LIN {X 0,Y 473.473,Z 413.056,A -85,B 0,C 180,E1 -7449.691,E2 -7449.691} C_VEL
LIN {X 0,Y 472.779,Z 426.431,A -85,B 0,C 180,E1 -7450.347,E2 -7450.347} C_VEL
LIN {X 0,Y 472.019,Z 440.423,A -85,B 0,C 180,E1 -7451.218,E2 -7451.218} C_VEL
LIN {X 0,Y 471.172,Z 453.208,A -85,B 0,C 180,E1 -7452.195,E2 -7452.195} C_VEL
LIN {X 0,Y 470.275,Z 466.134,A -85,B 0,C 180,E1 -7453.399,E2 -7453.399} C_VEL
LIN {X 0,Y 469.524,Z 476.835,A -85,B 0,C 180,E1 -7454.593,E2 -7454.593} C_VEL
LIN {X 0,Y 468.86,Z 486.774,A -85,B 0,C 180,E1 -7455.902,E2 -7455.902} C_VEL
LIN {X 0,Y 468.161,Z 496.122,A -85,B 0,C 180,E1 -7457.363,E2 -7457.363} C_VEL
LIN {X 0,Y 467.712,Z 504.564,A -85,B 0,C 180,E1 -7458.955,E2 -7458.955} C_VEL
LIN {X 0,Y 467.282,Z 511.235,A -85,B 0,C 180,E1 -7460.477,E2 -7460.477} C_VEL
LIN {X 0,Y 467.004,Z 517.412,A -85,B 0,C 180,E1 -7462.216,E2 -7462.216} C_VEL
LIN {X 0,Y 466.887,Z 522.181,A -85,B 0,C 180,E1 -7463.952,E2 -7463.952} C_VEL
LIN {X 0,Y 466.68,Z 525.681,A -85,B 0,C 180,E1 -7465.682,E2 -7465.682} C_VEL
LIN {X 0,Y 466.678,Z 527.994,A -85,B 0,C 180,E1 -7467.411,E2 -7467.411} C_VEL
LIN {X 0,Y 466.616,Z 529.179,A -85,B 0,C 180,E1 -7469.137,E2 -7469.137} C_VEL
LIN {X 0,Y 466.617,Z 529.196,A -85,B 0,C 180,E1 -7470.863,E2 -7470.863} C_VEL
LIN {X 0,Y 466.678,Z 528.081,A -85,B 0,C 180,E1 -7472.589,E2 -7472.589} C_VEL
LIN {X 0,Y 466.678,Z 525.836,A -85,B 0,C 180,E1 -7474.318,E2 -7474.318} C_VEL
LIN {X 0,Y 466.867,Z 522.401,A -85,B 0,C 180,E1 -7476.049,E2 -7476.049} C_VEL
LIN {X 0,Y 467.003,Z 517.703,A -85,B 0,C 180,E1 -7477.784,E2 -7477.784} C_VEL
LIN {X 0,Y 467.26,Z 511.612,A -85,B 0,C 180,E1 -7479.523,E2 -7479.523} C_VEL
LIN {X 0,Y 467.793,Z 503.938,A -85,B 0,C 180,E1 -7481.262,E2 -7481.262} C_VEL
LIN {X 0,Y 468.244,Z 495.615,A -85,B 0,C 180,E1 -7482.815,E2 -7482.815} C_VEL
LIN {X 0,Y 468.908,Z 485.901,A -85,B 0,C 180,E1 -7484.318,E2 -7484.318} C_VEL
LIN {X 0,Y 469.626,Z 475.791,A -85,B 0,C 180,E1 -7485.627,E2 -7485.627} C_VEL
LIN {X 0,Y 470.422,Z 464.385,A -85,B 0,C 180,E1 -7486.871,E2 -7486.871} C_VEL
LIN {X 0,Y 471.307,Z 451.682,A -85,B 0,C 180,E1 -7488.024,E2 -7488.024} C_VEL
LIN {X 0,Y 472.142,Z 438.564,A -85,B 0,C 180,E1 -7489.002,E2 -7489.002} C_VEL
LIN {X 0,Y 472.815,Z 426.069,A -85,B 0,C 180,E1 -7489.764,E2 -7489.764} C_VEL
LIN {X 0,Y 473.535,Z 411.357,A -85,B 0,C 180,E1 -7490.473,E2 -7490.473} C_VEL
LIN {X 0,Y 474.056,Z 395.831,A -85,B 0,C 180,E1 -7491.026,E2 -7491.026} C_VEL
LIN {X 0,Y 474.436,Z 382.034,A -85,B 0,C 180,E1 -7491.359,E2 -7491.359} C_VEL
LIN {X 0,Y 475.776,Z 266.855,A -85,B 0,C 180,E1 -7493.153,E2 -7493.153} C_VEL
LIN {X 0,Y 475.977,Z 239.419,A -85,B 0,C 180,E1 -7493.585,E2 -7493.585} C_VEL
LIN {X 0,Y 471.515,Z 220.798,A -85,B 0,C 180,E1 -7494.128,E2 -7494.128} C_VEL
LIN {X 0,Y 471.131,Z 219.52,A -85,B 0,C 180,E1 -7494.183,E2 -7494.183} C_VEL
LIN {X 0,Y 467.685,Z 203.856,A -85,B 0,C 180,E1 -7497.16,E2 -7497.16} C_VEL
LIN {X 0,Y 467.568,Z 203.868,A -85,B 0,C 180,E1 -7500.733,E2 -7500.733} C_VEL
LIN {X 0,Y 467.585,Z 203.866,A -85,B 0,C 180,E1 -7503.787,E2 -7503.787} C_VEL
LIN {X 0,Y 467.547,Z 203.87,A -85,B 0,C 180,E1 -7507.186,E2 -7507.186} C_VEL
LIN {X 0,Y 467.575,Z 203.862,A -85,B 0,C 180,E1 -7510.264,E2 -7510.264} C_VEL
LIN {X 0,Y 467.583,Z 203.863,A -85,B 0,C 180,E1 -7512.566,E2 -7512.566} C_VEL
LIN {X 0,Y 467.566,Z 203.868,A -85,B 0,C 180,E1 -7515.052,E2 -7515.052} C_VEL
LIN {X 0,Y 467.584,Z 203.86,A -85,B 0,C 180,E1 -7517.439,E2 -7517.439} C_VEL
LIN {X 0,Y 467.607,Z 203.863,A -85,B 0,C 180,E1 -7520.858,E2 -7520.858} C_VEL
LIN {X 0,Y 467.557,Z 203.864,A -85,B 0,C 180,E1 -7524.26,E2 -7524.26} C_VEL
LIN {X 0,Y 467.576,Z 203.858,A -85,B 0,C 180,E1 -7527.32,E2 -7527.32} C_VEL
LIN {X 0,Y 467.571,Z 203.863,A -85,B 0,C 180,E1 -7530.665,E2 -7530.665} C_VEL
LIN {X 0,Y 467.609,Z 203.861,A -85,B 0,C 180,E1 -7533.199,E2 -7533.199} C_VEL
LIN {X 0,Y 467.585,Z 203.864,A -85,B 0,C 180,E1 -7536.468,E2 -7536.468} C_VEL
LIN {X 0,Y 467.615,Z 203.858,A -85,B 0,C 180,E1 -7539.777,E2 -7539.777} C_VEL
LIN {X 0,Y 467.601,Z 203.86,A -85,B 0,C 180,E1 -7542.506,E2 -7542.506} C_VEL
LIN {X 0,Y 467.598,Z 203.859,A -85,B 0,C 180,E1 -7545.196,E2 -7545.196} C_VEL
LIN {X 0,Y 467.648,Z 203.854,A -85,B 0,C 180,E1 -7547.854,E2 -7547.854} C_VEL
LIN {X 0,Y 467.673,Z 203.852,A -85,B 0,C 180,E1 -7551.357,E2 -7551.357} C_VEL
LIN {X 0,Y 467.735,Z 203.842,A -85,B 0,C 180,E1 -7553.962,E2 -7553.962} C_VEL
LIN {X 0,Y 467.851,Z 203.829,A -85,B 0,C 180,E1 -7557.417,E2 -7557.417} C_VEL
LIN {X 0,Y 467.872,Z 203.822,A -85,B 0,C 180,E1 -7560,E2 -7560} C_VEL
LIN {X 0,Y 467.851,Z 203.834,A -85,B 0,C 180,E1 -7562.583,E2 -7562.583} C_VEL
LIN {X 0,Y 467.735,Z 203.845,A -85,B 0,C 180,E1 -7566.037,E2 -7566.037} C_VEL
LIN {X 0,Y 467.673,Z 203.853,A -85,B 0,C 180,E1 -7568.643,E2 -7568.643} C_VEL
LIN {X 0,Y 467.647,Z 203.858,A -85,B 0,C 180,E1 -7572.146,E2 -7572.146} C_VEL
LIN {X 0,Y 467.646,Z 203.856,A -85,B 0,C 180,E1 -7575.695,E2 -7575.695} C_VEL
LIN {X 0,Y 467.609,Z 203.864,A -85,B 0,C 180,E1 -7578.765,E2 -7578.765} C_VEL
LIN {X 0,Y 467.572,Z 203.861,A -85,B 0,C 180,E1 -7581.269,E2 -7581.269} C_VEL
LIN {X 0,Y 467.565,Z 203.869,A -85,B 0,C 180,E1 -7583.944,E2 -7583.944} C_VEL
LIN {X 0,Y 467.608,Z 203.862,A -85,B 0,C 180,E1 -7586.801,E2 -7586.801} C_VEL
LIN {X 0,Y 467.58,Z 203.865,A -85,B 0,C 180,E1 -7589.736,E2 -7589.736} C_VEL
LIN {X 0,Y 467.576,Z 203.862,A -85,B 0,C 180,E1 -7592.759,E2 -7592.759} C_VEL
LIN {X 0,Y 467.55,Z 203.871,A -85,B 0,C 180,E1 -7595.89,E2 -7595.89} C_VEL
LIN {X 0,Y 467.575,Z 203.86,A -85,B 0,C 180,E1 -7599.145,E2 -7599.145} C_VEL
LIN {X 0,Y 467.58,Z 203.865,A -85,B 0,C 180,E1 -7602.568,E2 -7602.568} C_VEL
LIN {X 0,Y 467.565,Z 203.865,A -85,B 0,C 180,E1 -7605.054,E2 -7605.054} C_VEL
LIN {X 0,Y 467.584,Z 203.864,A -85,B 0,C 180,E1 -7607.441,E2 -7607.441} C_VEL
LIN {X 0,Y 467.595,Z 203.861,A -85,B 0,C 180,E1 -7610.858,E2 -7610.858} C_VEL
LIN {X 0,Y 467.559,Z 203.869,A -85,B 0,C 180,E1 -7614.261,E2 -7614.261} C_VEL
LIN {X 0,Y 467.579,Z 203.868,A -85,B 0,C 180,E1 -7617.321,E2 -7617.321} C_VEL
LIN {X 0,Y 467.595,Z 203.901,A -85,B 0,C 180,E1 -7619.613,E2 -7619.613} C_VEL
LIN {X 0,Y 471.126,Z 218.42,A -85,B 0,C 180,E1 -7622.104,E2 -7622.104} C_VEL
LIN {X 0,Y 472.237,Z 223.722,A -85,B 0,C 180,E1 -7622.979,E2 -7622.979} C_VEL
LIN {X 0,Y 471.169,Z 243.147,A -85,B 0,C 180,E1 -7625.855,E2 -7625.855} C_VEL
LIN {X 0,Y 475.907,Z 268.042,A -85,B 0,C 180,E1 -7626.52,E2 -7626.52} C_VEL
LIN {X 0,Y 474.175,Z 410.193,A -85,B 0,C 180,E1 -7628.737,E2 -7628.737} C_VEL
LIN {X 0,Y 473.629,Z 425.893,A -85,B 0,C 180,E1 -7629.16,E2 -7629.16} C_VEL
LIN {X 0,Y 473.043,Z 439.94,A -85,B 0,C 180,E1 -7629.702,E2 -7629.702} C_VEL
LIN {X 0,Y 472.253,Z 454.431,A -85,B 0,C 180,E1 -7630.438,E2 -7630.438} C_VEL
LIN {X 0,Y 471.47,Z 467.941,A -85,B 0,C 180,E1 -7631.308,E2 -7631.308} C_VEL
LIN {X 0,Y 470.494,Z 481.695,A -85,B 0,C 180,E1 -7632.394,E2 -7632.394} C_VEL
LIN {X 0,Y 469.7,Z 494.151,A -85,B 0,C 180,E1 -7633.596,E2 -7633.596} C_VEL
LIN {X 0,Y 468.813,Z 506.366,A -85,B 0,C 180,E1 -7635.014,E2 -7635.014} C_VEL
LIN {X 0,Y 468.101,Z 517.231,A -85,B 0,C 180,E1 -7636.543,E2 -7636.543} C_VEL
LIN {X 0,Y 467.611,Z 526.284,A -85,B 0,C 180,E1 -7638.074,E2 -7638.074} C_VEL
LIN {X 0,Y 467.228,Z 533.793,A -85,B 0,C 180,E1 -7639.601,E2 -7639.601} C_VEL
LIN {X 0,Y 466.908,Z 540.8,A -85,B 0,C 180,E1 -7641.343,E2 -7641.343} C_VEL
LIN {X 0,Y 466.818,Z 546.314,A -85,B 0,C 180,E1 -7643.083,E2 -7643.083} C_VEL
LIN {X 0,Y 466.684,Z 550.48,A -85,B 0,C 180,E1 -7644.816,E2 -7644.816} C_VEL
LIN {X 0,Y 466.634,Z 553.402,A -85,B 0,C 180,E1 -7646.546,E2 -7646.546} C_VEL
LIN {X 0,Y 466.604,Z 555.144,A -85,B 0,C 180,E1 -7648.274,E2 -7648.274} C_VEL
LIN {X 0,Y 466.595,Z 555.742,A -85,B 0,C 180,E1 -7650,E2 -7650} C_VEL
LIN {X 0,Y 466.604,Z 555.142,A -85,B 0,C 180,E1 -7651.726,E2 -7651.726} C_VEL
LIN {X 0,Y 466.634,Z 553.396,A -85,B 0,C 180,E1 -7653.454,E2 -7653.454} C_VEL
LIN {X 0,Y 466.688,Z 550.477,A -85,B 0,C 180,E1 -7655.184,E2 -7655.184} C_VEL
LIN {X 0,Y 466.821,Z 546.316,A -85,B 0,C 180,E1 -7656.917,E2 -7656.917} C_VEL
LIN {X 0,Y 466.908,Z 540.799,A -85,B 0,C 180,E1 -7658.657,E2 -7658.657} C_VEL
LIN {X 0,Y 467.228,Z 533.783,A -85,B 0,C 180,E1 -7660.399,E2 -7660.399} C_VEL
LIN {X 0,Y 467.592,Z 526.274,A -85,B 0,C 180,E1 -7661.927,E2 -7661.927} C_VEL
LIN {X 0,Y 468.076,Z 517.225,A -85,B 0,C 180,E1 -7663.457,E2 -7663.457} C_VEL
LIN {X 0,Y 468.816,Z 506.356,A -85,B 0,C 180,E1 -7664.986,E2 -7664.986} C_VEL
LIN {X 0,Y 469.668,Z 494.142,A -85,B 0,C 180,E1 -7666.406,E2 -7666.406} C_VEL
LIN {X 0,Y 470.535,Z 481.688,A -85,B 0,C 180,E1 -7667.605,E2 -7667.605} C_VEL
LIN {X 0,Y 471.412,Z 469.438,A -85,B 0,C 180,E1 -7668.582,E2 -7668.582} C_VEL
LIN {X 0,Y 472.163,Z 456.21,A -85,B 0,C 180,E1 -7669.453,E2 -7669.453} C_VEL
LIN {X 0,Y 472.927,Z 443.069,A -85,B 0,C 180,E1 -7670.146,E2 -7670.146} C_VEL
LIN {X 0,Y 473.573,Z 427.912,A -85,B 0,C 180,E1 -7670.766,E2 -7670.766} C_VEL
LIN {X 0,Y 474.066,Z 412.397,A -85,B 0,C 180,E1 -7671.212,E2 -7671.212} C_VEL
LIN {X 0,Y 474.424,Z 390.321,A -85,B 0,C 180,E1 -7671.594,E2 -7671.594} C_VEL
LIN {X 0,Y 475.907,Z 267.885,A -85,B 0,C 180,E1 -7673.48,E2 -7673.48} C_VEL
LIN {X 0,Y 471.138,Z 243.171,A -85,B 0,C 180,E1 -7674.139,E2 -7674.139} C_VEL
LIN {X 0,Y 472.159,Z 225.592,A -85,B 0,C 180,E1 -7676.736,E2 -7676.736} C_VEL
LIN {X 0,Y 471.99,Z 222.192,A -85,B 0,C 180,E1 -7677.264,E2 -7677.264} C_VEL
LIN {X 0,Y 468.627,Z 208.028,A -85,B 0,C 180,E1 -7679.662,E2 -7679.662} C_VEL
LIN {X 0,Y 467.557,Z 203.866,A -85,B 0,C 180,E1 -7680.421,E2 -7680.421} C_VEL
LIN {X 0,Y 467.58,Z 203.857,A -85,B 0,C 180,E1 -7682.758,E2 -7682.758} C_VEL
LIN {X 0,Y 467.552,Z 203.869,A -85,B 0,C 180,E1 -7685.889,E2 -7685.889} C_VEL
LIN {X 0,Y 467.595,Z 203.862,A -85,B 0,C 180,E1 -7689.142,E2 -7689.142} C_VEL
LIN {X 0,Y 467.581,Z 203.863,A -85,B 0,C 180,E1 -7692.566,E2 -7692.566} C_VEL
LIN {X 0,Y 467.565,Z 203.863,A -85,B 0,C 180,E1 -7695.052,E2 -7695.052} C_VEL
LIN {X 0,Y 467.583,Z 203.862,A -85,B 0,C 180,E1 -7697.439,E2 -7697.439} C_VEL
LIN {X 0,Y 467.593,Z 203.859,A -85,B 0,C 180,E1 -7700.856,E2 -7700.856} C_VEL
LIN {X 0,Y 467.556,Z 203.865,A -85,B 0,C 180,E1 -7704.26,E2 -7704.26} C_VEL
LIN {X 0,Y 467.575,Z 203.861,A -85,B 0,C 180,E1 -7707.32,E2 -7707.32} C_VEL
LIN {X 0,Y 467.57,Z 203.862,A -85,B 0,C 180,E1 -7710.665,E2 -7710.665} C_VEL
LIN {X 0,Y 467.608,Z 203.859,A -85,B 0,C 180,E1 -7713.199,E2 -7713.199} C_VEL
LIN {X 0,Y 467.584,Z 203.858,A -85,B 0,C 180,E1 -7716.468,E2 -7716.468} C_VEL
LIN {X 0,Y 467.615,Z 203.857,A -85,B 0,C 180,E1 -7719.777,E2 -7719.777} C_VEL
LIN {X 0,Y 467.6,Z 203.859,A -85,B 0,C 180,E1 -7722.507,E2 -7722.507} C_VEL
LIN {X 0,Y 467.597,Z 203.862,A -85,B 0,C 180,E1 -7725.196,E2 -7725.196} C_VEL
LIN {X 0,Y 467.647,Z 203.857,A -85,B 0,C 180,E1 -7727.854,E2 -7727.854} C_VEL
LIN {X 0,Y 467.673,Z 203.854,A -85,B 0,C 180,E1 -7731.357,E2 -7731.357} C_VEL
LIN {X 0,Y 467.735,Z 203.845,A -85,B 0,C 180,E1 -7733.963,E2 -7733.963} C_VEL
LIN {X 0,Y 467.851,Z 203.835,A -85,B 0,C 180,E1 -7737.417,E2 -7737.417} C_VEL
LIN {X 0,Y 467.873,Z 203.824,A -85,B 0,C 180,E1 -7740,E2 -7740} C_VEL
LIN {X 0,Y 467.851,Z 203.829,A -85,B 0,C 180,E1 -7742.583,E2 -7742.583} C_VEL
LIN {X 0,Y 467.738,Z 203.843,A -85,B 0,C 180,E1 -7746.038,E2 -7746.038} C_VEL
LIN {X 0,Y 467.674,Z 203.849,A -85,B 0,C 180,E1 -7748.643,E2 -7748.643} C_VEL
LIN {X 0,Y 467.648,Z 203.852,A -85,B 0,C 180,E1 -7752.146,E2 -7752.146} C_VEL
LIN {X 0,Y 467.63,Z 203.856,A -85,B 0,C 180,E1 -7755.695,E2 -7755.695} C_VEL
LIN {X 0,Y 467.609,Z 203.862,A -85,B 0,C 180,E1 -7758.765,E2 -7758.765} C_VEL
LIN {X 0,Y 467.572,Z 203.868,A -85,B 0,C 180,E1 -7761.269,E2 -7761.269} C_VEL
LIN {X 0,Y 467.565,Z 203.862,A -85,B 0,C 180,E1 -7763.944,E2 -7763.944} C_VEL
LIN {X 0,Y 467.608,Z 203.849,A -85,B 0,C 180,E1 -7766.801,E2 -7766.801} C_VEL
LIN {X 0,Y 467.581,Z 203.863,A -85,B 0,C 180,E1 -7769.736,E2 -7769.736} C_VEL
LIN {X 0,Y 467.577,Z 203.868,A -85,B 0,C 180,E1 -7772.759,E2 -7772.759} C_VEL
LIN {X 0,Y 467.551,Z 203.865,A -85,B 0,C 180,E1 -7775.89,E2 -7775.89} C_VEL
LIN {X 0,Y 467.577,Z 203.864,A -85,B 0,C 180,E1 -7779.145,E2 -7779.145} C_VEL
LIN {X 0,Y 467.582,Z 203.864,A -85,B 0,C 180,E1 -7782.568,E2 -7782.568} C_VEL
LIN {X 0,Y 467.567,Z 203.869,A -85,B 0,C 180,E1 -7785.054,E2 -7785.054} C_VEL
LIN {X 0,Y 467.585,Z 203.864,A -85,B 0,C 180,E1 -7787.441,E2 -7787.441} C_VEL
LIN {X 0,Y 467.579,Z 203.864,A -85,B 0,C 180,E1 -7790.856,E2 -7790.856} C_VEL
LIN {X 0,Y 467.557,Z 203.867,A -85,B 0,C 180,E1 -7794.262,E2 -7794.262} C_VEL
LIN {X 0,Y 467.58,Z 203.866,A -85,B 0,C 180,E1 -7797.322,E2 -7797.322} C_VEL
LIN {X 0,Y 467.569,Z 203.868,A -85,B 0,C 180,E1 -7800.668,E2 -7800.668} C_VEL
LIN {X 0,Y 467.686,Z 203.923,A -85,B 0,C 180,E1 -7802.952,E2 -7802.952} C_VEL
LIN {X 0,Y 470.94,Z 218.784,A -85,B 0,C 180,E1 -7805.771,E2 -7805.771} C_VEL
LIN {X 0,Y 471.099,Z 219.687,A -85,B 0,C 180,E1 -7805.924,E2 -7805.924} C_VEL
LIN {X 0,Y 473.398,Z 228.223,A -85,B 0,C 180,E1 -7806.189,E2 -7806.189} C_VEL
LIN {X 0,Y 476.069,Z 240.442,A -85,B 0,C 180,E1 -7806.53,E2 -7806.53} C_VEL
LIN {X 0,Y 475.647,Z 279.036,A -85,B 0,C 180,E1 -7807.129,E2 -7807.129} C_VEL
LIN {X 0,Y 475.039,Z 284.883,A -85,B 0,C 180,E1 -7807.192,E2 -7807.192} C_VEL
LIN {X 0,Y 469.524,Z 303.949,A -85,B 0,C 180,E1 -7807.216,E2 -7807.216} C_VEL
LIN {X 0,Y 468.797,Z 309.804,A -85,B 0,C 180,E1 -7807.274,E2 -7807.274} C_VEL
LIN {X 0,Y 467.794,Z 384.871,A -85,B 0,C 180,E1 -7808.467,E2 -7808.467} C_VEL
LIN {X 0,Y 467.377,Z 400.309,A -85,B 0,C 180,E1 -7808.888,E2 -7808.888} C_VEL
LIN {X 0,Y 466.813,Z 413.523,A -85,B 0,C 180,E1 -7809.399,E2 -7809.399} C_VEL
LIN {X 0,Y 466.116,Z 426.64,A -85,B 0,C 180,E1 -7810.054,E2 -7810.054} C_VEL
LIN {X 0,Y 465.29,Z 440.631,A -85,B 0,C 180,E1 -7810.936,E2 -7810.936} C_VEL
LIN {X 0,Y 464.382,Z 453.415,A -85,B 0,C 180,E1 -7811.926,E2 -7811.926} C_VEL
LIN {X 0,Y 463.524,Z 465.627,A -85,B 0,C 180,E1 -7813.074,E2 -7813.074} C_VEL
LIN {X 0,Y 462.659,Z 477.04,A -85,B 0,C 180,E1 -7814.358,E2 -7814.358} C_VEL
LIN {X 0,Y 461.948,Z 486.979,A -85,B 0,C 180,E1 -7815.687,E2 -7815.687} C_VEL
LIN {X 0,Y 461.146,Z 496.829,A -85,B 0,C 180,E1 -7817.26,E2 -7817.26} C_VEL
LIN {X 0,Y 460.731,Z 504.767,A -85,B 0,C 180,E1 -7818.785,E2 -7818.785} C_VEL
LIN {X 0,Y 460.259,Z 511.438,A -85,B 0,C 180,E1 -7820.331,E2 -7820.331} C_VEL
LIN {X 0,Y 459.963,Z 517.614,A -85,B 0,C 180,E1 -7822.096,E2 -7822.096} C_VEL
LIN {X 0,Y 459.816,Z 522.383,A -85,B 0,C 180,E1 -7823.858,E2 -7823.858} C_VEL
LIN {X 0,Y 459.594,Z 525.883,A -85,B 0,C 180,E1 -7825.615,E2 -7825.615} C_VEL
LIN {X 0,Y 459.6,Z 528.195,A -85,B 0,C 180,E1 -7827.371,E2 -7827.371} C_VEL
LIN {X 0,Y 459.52,Z 529.38,A -85,B 0,C 180,E1 -7829.124,E2 -7829.124} C_VEL
LIN {X 0,Y 459.521,Z 529.397,A -85,B 0,C 180,E1 -7830.876,E2 -7830.876} C_VEL
LIN {X 0,Y 459.6,Z 528.281,A -85,B 0,C 180,E1 -7832.629,E2 -7832.629} C_VEL
LIN {X 0,Y 459.592,Z 526.037,A -85,B 0,C 180,E1 -7834.385,E2 -7834.385} C_VEL
LIN {X 0,Y 459.794,Z 522.602,A -85,B 0,C 180,E1 -7836.142,E2 -7836.142} C_VEL
LIN {X 0,Y 459.962,Z 517.902,A -85,B 0,C 180,E1 -7837.904,E2 -7837.904} C_VEL
LIN {X 0,Y 460.231,Z 511.812,A -85,B 0,C 180,E1 -7839.67,E2 -7839.67} C_VEL
LIN {X 0,Y 460.8,Z 504.137,A -85,B 0,C 180,E1 -7841.436,E2 -7841.436} C_VEL
LIN {X 0,Y 461.26,Z 496.054,A -85,B 0,C 180,E1 -7842.97,E2 -7842.97} C_VEL
LIN {X 0,Y 461.994,Z 486.1,A -85,B 0,C 180,E1 -7844.537,E2 -7844.537} C_VEL
LIN {X 0,Y 462.737,Z 475.99,A -85,B 0,C 180,E1 -7845.865,E2 -7845.865} C_VEL
LIN {X 0,Y 463.578,Z 465.088,A -85,B 0,C 180,E1 -7847.073,E2 -7847.073} C_VEL
LIN {X 0,Y 464.459,Z 453.163,A -85,B 0,C 180,E1 -7848.185,E2 -7848.185} C_VEL
LIN {X 0,Y 465.312,Z 440.334,A -85,B 0,C 180,E1 -7849.178,E2 -7849.178} C_VEL
LIN {X 0,Y 466.155,Z 426.261,A -85,B 0,C 180,E1 -7850.059,E2 -7850.059} C_VEL
LIN {X 0,Y 466.902,Z 411.121,A -85,B 0,C 180,E1 -7850.796,E2 -7850.796} C_VEL
LIN {X 0,Y 467.477,Z 395.646,A -85,B 0,C 180,E1 -7851.349,E2 -7851.349} C_VEL
LIN {X 0,Y 467.857,Z 381.93,A -85,B 0,C 180,E1 -7851.68,E2 -7851.68} C_VEL
LIN {X 0,Y 469.426,Z 255.668,A -85,B 0,C 180,E1 -7853.67,E2 -7853.67} C_VEL
LIN {X 0,Y 469.433,Z 240.217,A -85,B 0,C 180,E1 -7853.923,E2 -7853.923} C_VEL
LIN {X 0,Y 465.221,Z 222.931,A -85,B 0,C 180,E1 -7854.443,E2 -7854.443} C_VEL
LIN {X 0,Y 463.984,Z 219.732,A -85,B 0,C 180,E1 -7854.58,E2 -7854.58} C_VEL
LIN {X 0,Y 460.94,Z 206.042,A -85,B 0,C 180,E1 -7857.22,E2 -7857.22} C_VEL
LIN {X 0,Y 460.592,Z 204.74,A -85,B 0,C 180,E1 -7857.491,E2 -7857.491} C_VEL
LIN {X 0,Y 460.509,Z 204.747,A -85,B 0,C 180,E1 -7860.239,E2 -7860.239} C_VEL
LIN {X 0,Y 460.527,Z 204.749,A -85,B 0,C 180,E1 -7863.324,E2 -7863.324} C_VEL
LIN {X 0,Y 460.475,Z 204.749,A -85,B 0,C 180,E1 -7866.528,E2 -7866.528} C_VEL
LIN {X 0,Y 460.542,Z 204.745,A -85,B 0,C 180,E1 -7868.897,E2 -7868.897} C_VEL
LIN {X 0,Y 460.52,Z 204.743,A -85,B 0,C 180,E1 -7872.18,E2 -7872.18} C_VEL
LIN {X 0,Y 460.512,Z 204.749,A -85,B 0,C 180,E1 -7875.411,E2 -7875.411} C_VEL
LIN {X 0,Y 460.53,Z 204.737,A -85,B 0,C 180,E1 -7878.396,E2 -7878.396} C_VEL
LIN {X 0,Y 460.536,Z 204.739,A -85,B 0,C 180,E1 -7881.268,E2 -7881.268} C_VEL
LIN {X 0,Y 460.508,Z 204.743,A -85,B 0,C 180,E1 -7884.554,E2 -7884.554} C_VEL
LIN {X 0,Y 460.526,Z 204.732,A -85,B 0,C 180,E1 -7887.715,E2 -7887.715} C_VEL
LIN {X 0,Y 460.54,Z 204.739,A -85,B 0,C 180,E1 -7890.769,E2 -7890.769} C_VEL
LIN {X 0,Y 460.555,Z 204.736,A -85,B 0,C 180,E1 -7893.734,E2 -7893.734} C_VEL
LIN {X 0,Y 460.538,Z 204.743,A -85,B 0,C 180,E1 -7896.623,E2 -7896.623} C_VEL
LIN {X 0,Y 460.544,Z 204.741,A -85,B 0,C 180,E1 -7899.452,E2 -7899.452} C_VEL
LIN {X 0,Y 460.551,Z 204.736,A -85,B 0,C 180,E1 -7902.23,E2 -7902.23} C_VEL
LIN {X 0,Y 460.557,Z 204.739,A -85,B 0,C 180,E1 -7904.964,E2 -7904.964} C_VEL
LIN {X 0,Y 460.604,Z 204.736,A -85,B 0,C 180,E1 -7908.559,E2 -7908.559} C_VEL
LIN {X 0,Y 460.686,Z 204.722,A -85,B 0,C 180,E1 -7912.108,E2 -7912.108} C_VEL
LIN {X 0,Y 460.689,Z 204.722,A -85,B 0,C 180,E1 -7914.748,E2 -7914.748} C_VEL
LIN {X 0,Y 460.816,Z 204.706,A -85,B 0,C 180,E1 -7917.377,E2 -7917.377} C_VEL
LIN {X 0,Y 460.843,Z 204.698,A -85,B 0,C 180,E1 -7920,E2 -7920} C_VEL
LIN {X 0,Y 460.816,Z 204.71,A -85,B 0,C 180,E1 -7922.622,E2 -7922.622} C_VEL
LIN {X 0,Y 460.701,Z 204.722,A -85,B 0,C 180,E1 -7926.13,E2 -7926.13} C_VEL
LIN {X 0,Y 460.62,Z 204.732,A -85,B 0,C 180,E1 -7928.776,E2 -7928.776} C_VEL
LIN {X 0,Y 460.604,Z 204.735,A -85,B 0,C 180,E1 -7932.445,E2 -7932.445} C_VEL
LIN {X 0,Y 460.613,Z 204.735,A -85,B 0,C 180,E1 -7936.007,E2 -7936.007} C_VEL
LIN {X 0,Y 460.561,Z 204.739,A -85,B 0,C 180,E1 -7939.616,E2 -7939.616} C_VEL
LIN {X 0,Y 460.503,Z 204.749,A -85,B 0,C 180,E1 -7942.429,E2 -7942.429} C_VEL
LIN {X 0,Y 460.559,Z 204.737,A -85,B 0,C 180,E1 -7945.802,E2 -7945.802} C_VEL
LIN {X 0,Y 460.55,Z 204.745,A -85,B 0,C 180,E1 -7948.233,E2 -7948.233} C_VEL
LIN {X 0,Y 460.517,Z 204.743,A -85,B 0,C 180,E1 -7951.284,E2 -7951.284} C_VEL
LIN {X 0,Y 460.527,Z 204.745,A -85,B 0,C 180,E1 -7954.507,E2 -7954.507} C_VEL
LIN {X 0,Y 460.495,Z 204.747,A -85,B 0,C 180,E1 -7957.624,E2 -7957.624} C_VEL
LIN {X 0,Y 460.535,Z 204.732,A -85,B 0,C 180,E1 -7960.27,E2 -7960.27} C_VEL
LIN {X 0,Y 460.494,Z 204.747,A -85,B 0,C 180,E1 -7963.376,E2 -7963.376} C_VEL
LIN {X 0,Y 460.495,Z 204.747,A -85,B 0,C 180,E1 -7966.625,E2 -7966.625} C_VEL
LIN {X 0,Y 460.553,Z 204.743,A -85,B 0,C 180,E1 -7969.729,E2 -7969.729} C_VEL
LIN {X 0,Y 460.524,Z 204.739,A -85,B 0,C 180,E1 -7972.52,E2 -7972.52} C_VEL
LIN {X 0,Y 460.545,Z 204.745,A -85,B 0,C 180,E1 -7975.625,E2 -7975.625} C_VEL
LIN {X 0,Y 460.534,Z 204.742,A -85,B 0,C 180,E1 -7978.745,E2 -7978.745} C_VEL
LIN {X 0,Y 460.566,Z 204.887,A -85,B 0,C 180,E1 -7979.289,E2 -7979.289} C_VEL
LIN {X 0,Y 464.003,Z 218.784,A -85,B 0,C 180,E1 -7981.726,E2 -7981.726} C_VEL
LIN {X 0,Y 465.427,Z 225.43,A -85,B 0,C 180,E1 -7982.846,E2 -7982.846} C_VEL
LIN {X 0,Y 464.373,Z 242.94,A -85,B 0,C 180,E1 -7985.478,E2 -7985.478} C_VEL
LIN {X 0,Y 469.382,Z 268.809,A -85,B 0,C 180,E1 -7986.189,E2 -7986.189} C_VEL
LIN {X 0,Y 467.581,Z 408.682,A -85,B 0,C 180,E1 -7988.393,E2 -7988.393} C_VEL
LIN {X 0,Y 467.101,Z 424.245,A -85,B 0,C 180,E1 -7988.804,E2 -7988.804} C_VEL
LIN {X 0,Y 466.417,Z 438.561,A -85,B 0,C 180,E1 -7989.348,E2 -7989.348} C_VEL
LIN {X 0,Y 465.651,Z 452.242,A -85,B 0,C 180,E1 -7990.034,E2 -7990.034} C_VEL
LIN {X 0,Y 464.751,Z 466.155,A -85,B 0,C 180,E1 -7990.913,E2 -7990.913} C_VEL
LIN {X 0,Y 463.845,Z 478.904,A -85,B 0,C 180,E1 -7991.905,E2 -7991.905} C_VEL
LIN {X 0,Y 462.924,Z 491.791,A -85,B 0,C 180,E1 -7993.12,E2 -7993.12} C_VEL
LIN {X 0,Y 462.119,Z 502.601,A -85,B 0,C 180,E1 -7994.339,E2 -7994.339} C_VEL
LIN {X 0,Y 461.427,Z 512.597,A -85,B 0,C 180,E1 -7995.67,E2 -7995.67} C_VEL
LIN {X 0,Y 460.768,Z 522.627,A -85,B 0,C 180,E1 -7997.268,E2 -7997.268} C_VEL
LIN {X 0,Y 460.392,Z 530.546,A -85,B 0,C 180,E1 -7998.777,E2 -7998.777} C_VEL
LIN {X 0,Y 459.939,Z 537.293,A -85,B 0,C 180,E1 -8000.324,E2 -8000.324} C_VEL
LIN {X 0,Y 459.765,Z 543.531,A -85,B 0,C 180,E1 -8002.093,E2 -8002.093} C_VEL
LIN {X 0,Y 459.617,Z 548.356,A -85,B 0,C 180,E1 -8003.856,E2 -8003.856} C_VEL
LIN {X 0,Y 459.517,Z 551.89,A -85,B 0,C 180,E1 -8005.614,E2 -8005.614} C_VEL
LIN {X 0,Y 459.573,Z 554.218,A -85,B 0,C 180,E1 -8007.371,E2 -8007.371} C_VEL
LIN {X 0,Y 459.519,Z 555.387,A -85,B 0,C 180,E1 -8009.124,E2 -8009.124} C_VEL
LIN {X 0,Y 459.519,Z 555.386,A -85,B 0,C 180,E1 -8010.876,E2 -8010.876} C_VEL
LIN {X 0,Y 459.573,Z 554.213,A -85,B 0,C 180,E1 -8012.629,E2 -8012.629} C_VEL
LIN {X 0,Y 459.517,Z 551.884,A -85,B 0,C 180,E1 -8014.386,E2 -8014.386} C_VEL
LIN {X 0,Y 459.64,Z 548.355,A -85,B 0,C 180,E1 -8016.144,E2 -8016.144} C_VEL
LIN {X 0,Y 459.765,Z 543.532,A -85,B 0,C 180,E1 -8017.907,E2 -8017.907} C_VEL
LIN {X 0,Y 459.939,Z 537.285,A -85,B 0,C 180,E1 -8019.676,E2 -8019.676} C_VEL
LIN {X 0,Y 460.392,Z 530.534,A -85,B 0,C 180,E1 -8021.223,E2 -8021.223} C_VEL
LIN {X 0,Y 460.733,Z 522.616,A -85,B 0,C 180,E1 -8022.733,E2 -8022.733} C_VEL
LIN {X 0,Y 461.429,Z 512.587,A -85,B 0,C 180,E1 -8024.329,E2 -8024.329} C_VEL
LIN {X 0,Y 462.137,Z 502.587,A -85,B 0,C 180,E1 -8025.66,E2 -8025.66} C_VEL
LIN {X 0,Y 462.948,Z 491.599,A -85,B 0,C 180,E1 -8026.898,E2 -8026.898} C_VEL
LIN {X 0,Y 463.866,Z 478.888,A -85,B 0,C 180,E1 -8028.095,E2 -8028.095} C_VEL
LIN {X 0,Y 464.807,Z 466.121,A -85,B 0,C 180,E1 -8029.085,E2 -8029.085} C_VEL
LIN {X 0,Y 465.667,Z 452.195,A -85,B 0,C 180,E1 -8029.966,E2 -8029.966} C_VEL
LIN {X 0,Y 466.424,Z 438.456,A -85,B 0,C 180,E1 -8030.654,E2 -8030.654} C_VEL
LIN {X 0,Y 467.087,Z 423.263,A -85,B 0,C 180,E1 -8031.226,E2 -8031.226} C_VEL
LIN {X 0,Y 467.579,Z 408.546,A -85,B 0,C 180,E1 -8031.607,E2 -8031.607} C_VEL
LIN {X 0,Y 469.38,Z 268.62,A -85,B 0,C 180,E1 -8033.811,E2 -8033.811} C_VEL
LIN {X 0,Y 464.401,Z 242.824,A -85,B 0,C 180,E1 -8034.533,E2 -8034.533} C_VEL
LIN {X 0,Y 465.383,Z 225.239,A -85,B 0,C 180,E1 -8037.181,E2 -8037.181} C_VEL
LIN {X 0,Y 462.596,Z 212.985,A -85,B 0,C 180,E1 -8039.272,E2 -8039.272} C_VEL
LIN {X 0,Y 460.544,Z 204.738,A -85,B 0,C 180,E1 -8040.744,E2 -8040.744} C_VEL
LIN {X 0,Y 460.526,Z 204.734,A -85,B 0,C 180,E1 -8043.324,E2 -8043.324} C_VEL
LIN {X 0,Y 460.475,Z 204.751,A -85,B 0,C 180,E1 -8046.529,E2 -8046.529} C_VEL
LIN {X 0,Y 460.57,Z 204.741,A -85,B 0,C 180,E1 -8049.857,E2 -8049.857} C_VEL
LIN {X 0,Y 460.508,Z 204.743,A -85,B 0,C 180,E1 -8052.9,E2 -8052.9} C_VEL
LIN {X 0,Y 460.506,Z 204.748,A -85,B 0,C 180,E1 -8055.83,E2 -8055.83} C_VEL
LIN {X 0,Y 460.533,Z 204.738,A -85,B 0,C 180,E1 -8058.989,E2 -8058.989} C_VEL
LIN {X 0,Y 460.533,Z 204.74,A -85,B 0,C 180,E1 -8061.268,E2 -8061.268} C_VEL
LIN {X 0,Y 460.507,Z 204.741,A -85,B 0,C 180,E1 -8064.554,E2 -8064.554} C_VEL
LIN {X 0,Y 460.525,Z 204.743,A -85,B 0,C 180,E1 -8067.715,E2 -8067.715} C_VEL
LIN {X 0,Y 460.539,Z 204.737,A -85,B 0,C 180,E1 -8070.769,E2 -8070.769} C_VEL
LIN {X 0,Y 460.555,Z 204.741,A -85,B 0,C 180,E1 -8073.734,E2 -8073.734} C_VEL
LIN {X 0,Y 460.538,Z 204.736,A -85,B 0,C 180,E1 -8076.624,E2 -8076.624} C_VEL
LIN {X 0,Y 460.543,Z 204.732,A -85,B 0,C 180,E1 -8079.452,E2 -8079.452} C_VEL
LIN {X 0,Y 460.55,Z 204.739,A -85,B 0,C 180,E1 -8082.23,E2 -8082.23} C_VEL
LIN {X 0,Y 460.556,Z 204.738,A -85,B 0,C 180,E1 -8084.965,E2 -8084.965} C_VEL
LIN {X 0,Y 460.604,Z 204.73,A -85,B 0,C 180,E1 -8088.559,E2 -8088.559} C_VEL
LIN {X 0,Y 460.686,Z 204.721,A -85,B 0,C 180,E1 -8092.108,E2 -8092.108} C_VEL
LIN {X 0,Y 460.689,Z 204.721,A -85,B 0,C 180,E1 -8094.748,E2 -8094.748} C_VEL
LIN {X 0,Y 460.816,Z 204.71,A -85,B 0,C 180,E1 -8097.378,E2 -8097.378} C_VEL
LIN {X 0,Y 460.844,Z 204.699,A -85,B 0,C 180,E1 -8100,E2 -8100} C_VEL
LIN {X 0,Y 460.816,Z 204.706,A -85,B 0,C 180,E1 -8102.623,E2 -8102.623} C_VEL
LIN {X 0,Y 460.704,Z 204.719,A -85,B 0,C 180,E1 -8106.13,E2 -8106.13} C_VEL
LIN {X 0,Y 460.621,Z 204.728,A -85,B 0,C 180,E1 -8108.776,E2 -8108.776} C_VEL
LIN {X 0,Y 460.604,Z 204.73,A -85,B 0,C 180,E1 -8112.445,E2 -8112.445} C_VEL
LIN {X 0,Y 460.592,Z 204.732,A -85,B 0,C 180,E1 -8115.998,E2 -8115.998} C_VEL
LIN {X 0,Y 460.562,Z 204.741,A -85,B 0,C 180,E1 -8118.902,E2 -8118.902} C_VEL
LIN {X 0,Y 460.508,Z 204.747,A -85,B 0,C 180,E1 -8121.486,E2 -8121.486} C_VEL
LIN {X 0,Y 460.535,Z 204.738,A -85,B 0,C 180,E1 -8124.333,E2 -8124.333} C_VEL
LIN {X 0,Y 460.572,Z 204.733,A -85,B 0,C 180,E1 -8127.244,E2 -8127.244} C_VEL
LIN {X 0,Y 460.52,Z 204.742,A -85,B 0,C 180,E1 -8130.239,E2 -8130.239} C_VEL
LIN {X 0,Y 460.523,Z 204.742,A -85,B 0,C 180,E1 -8133.325,E2 -8133.325} C_VEL
LIN {X 0,Y 460.473,Z 204.75,A -85,B 0,C 180,E1 -8136.53,E2 -8136.53} C_VEL
LIN {X 0,Y 460.54,Z 204.743,A -85,B 0,C 180,E1 -8138.898,E2 -8138.898} C_VEL
LIN {X 0,Y 460.518,Z 204.74,A -85,B 0,C 180,E1 -8142.182,E2 -8142.182} C_VEL
LIN {X 0,Y 460.516,Z 204.743,A -85,B 0,C 180,E1 -8145.413,E2 -8145.413} C_VEL
LIN {X 0,Y 460.532,Z 204.745,A -85,B 0,C 180,E1 -8148.398,E2 -8148.398} C_VEL
LIN {X 0,Y 460.523,Z 204.742,A -85,B 0,C 180,E1 -8151.268,E2 -8151.268} C_VEL
LIN {X 0,Y 460.508,Z 204.746,A -85,B 0,C 180,E1 -8154.555,E2 -8154.555} C_VEL
LIN {X 0,Y 460.53,Z 204.744,A -85,B 0,C 180,E1 -8157.716,E2 -8157.716} C_VEL
LIN {X 0,Y 460.539,Z 204.744,A -85,B 0,C 180,E1 -8160.77,E2 -8160.77} C_VEL
LIN {X 0,Y 460.632,Z 204.846,A -85,B 0,C 180,E1 -8162.636,E2 -8162.636} C_VEL
LIN {X 0,Y 463.971,Z 219.719,A -85,B 0,C 180,E1 -8165.509,E2 -8165.509} C_VEL
LIN {X 0,Y 466.373,Z 227.002,A -85,B 0,C 180,E1 -8165.783,E2 -8165.783} C_VEL
LIN {X 0,Y 469.585,Z 241.85,A -85,B 0,C 180,E1 -8166.205,E2 -8166.205} C_VEL
LIN {X 0,Y 468.797,Z 309.804,A -85,B 0,C 180,E1 -8167.274,E2 -8167.274} C_VEL
LIN {X 0,Y 468.085,Z 315.652,A -85,B 0,C 180,E1 -8167.333,E2 -8167.333} C_VEL
LIN {X 0,Y 462.565,Z 334.702,A -85,B 0,C 180,E1 -8167.358,E2 -8167.358} C_VEL
LIN {X 0,Y 461.855,Z 340.549,A -85,B 0,C 180,E1 -8167.418,E2 -8167.418} C_VEL
LIN {X 0,Y 461.205,Z 385.092,A -85,B 0,C 180,E1 -8168.144,E2 -8168.144} C_VEL
LIN {X 0,Y 460.764,Z 400.702,A -85,B 0,C 180,E1 -8168.576,E2 -8168.576} C_VEL
LIN {X 0,Y 460.157,Z 414.015,A -85,B 0,C 180,E1 -8169.1,E2 -8169.1} C_VEL
LIN {X 0,Y 459.313,Z 428.828,A -85,B 0,C 180,E1 -8169.863,E2 -8169.863} C_VEL
LIN {X 0,Y 458.472,Z 442.415,A -85,B 0,C 180,E1 -8170.757,E2 -8170.757} C_VEL
LIN {X 0,Y 457.531,Z 454.908,A -85,B 0,C 180,E1 -8171.762,E2 -8171.762} C_VEL
LIN {X 0,Y 456.701,Z 466.116,A -85,B 0,C 180,E1 -8172.844,E2 -8172.844} C_VEL
LIN {X 0,Y 455.776,Z 477.246,A -85,B 0,C 180,E1 -8174.116,E2 -8174.116} C_VEL
LIN {X 0,Y 455.047,Z 487.183,A -85,B 0,C 180,E1 -8175.465,E2 -8175.465} C_VEL
LIN {X 0,Y 454.258,Z 496.594,A -85,B 0,C 180,E1 -8176.982,E2 -8176.982} C_VEL
LIN {X 0,Y 453.749,Z 504.971,A -85,B 0,C 180,E1 -8178.611,E2 -8178.611} C_VEL
LIN {X 0,Y 453.239,Z 511.641,A -85,B 0,C 180,E1 -8180.179,E2 -8180.179} C_VEL
LIN {X 0,Y 452.912,Z 517.817,A -85,B 0,C 180,E1 -8181.972,E2 -8181.972} C_VEL
LIN {X 0,Y 452.731,Z 522.586,A -85,B 0,C 180,E1 -8183.762,E2 -8183.762} C_VEL
LIN {X 0,Y 452.513,Z 526.084,A -85,B 0,C 180,E1 -8185.546,E2 -8185.546} C_VEL
LIN {X 0,Y 452.525,Z 528.395,A -85,B 0,C 180,E1 -8187.33,E2 -8187.33} C_VEL
LIN {X 0,Y 452.428,Z 529.581,A -85,B 0,C 180,E1 -8189.11,E2 -8189.11} C_VEL
LIN {X 0,Y 452.428,Z 529.598,A -85,B 0,C 180,E1 -8190.89,E2 -8190.89} C_VEL
LIN {X 0,Y 452.525,Z 528.481,A -85,B 0,C 180,E1 -8192.67,E2 -8192.67} C_VEL
LIN {X 0,Y 452.511,Z 526.237,A -85,B 0,C 180,E1 -8194.454,E2 -8194.454} C_VEL
LIN {X 0,Y 452.71,Z 522.802,A -85,B 0,C 180,E1 -8196.238,E2 -8196.238} C_VEL
LIN {X 0,Y 452.911,Z 518.102,A -85,B 0,C 180,E1 -8198.028,E2 -8198.028} C_VEL
LIN {X 0,Y 453.211,Z 512.012,A -85,B 0,C 180,E1 -8199.821,E2 -8199.821} C_VEL
LIN {X 0,Y 453.789,Z 504.338,A -85,B 0,C 180,E1 -8201.615,E2 -8201.615} C_VEL
LIN {X 0,Y 454.286,Z 496.468,A -85,B 0,C 180,E1 -8203.133,E2 -8203.133} C_VEL
LIN {X 0,Y 455.093,Z 486.299,A -85,B 0,C 180,E1 -8204.762,E2 -8204.762} C_VEL
LIN {X 0,Y 455.86,Z 476.189,A -85,B 0,C 180,E1 -8206.111,E2 -8206.111} C_VEL
LIN {X 0,Y 456.716,Z 465.888,A -85,B 0,C 180,E1 -8207.272,E2 -8207.272} C_VEL
LIN {X 0,Y 457.684,Z 453.36,A -85,B 0,C 180,E1 -8208.464,E2 -8208.464} C_VEL
LIN {X 0,Y 458.606,Z 440.529,A -85,B 0,C 180,E1 -8209.469,E2 -8209.469} C_VEL
LIN {X 0,Y 459.504,Z 426.454,A -85,B 0,C 180,E1 -8210.362,E2 -8210.362} C_VEL
LIN {X 0,Y 460.254,Z 411.779,A -85,B 0,C 180,E1 -8211.089,E2 -8211.089} C_VEL
LIN {X 0,Y 460.845,Z 396.642,A -85,B 0,C 180,E1 -8211.645,E2 -8211.645} C_VEL
LIN {X 0,Y 461.269,Z 382.088,A -85,B 0,C 180,E1 -8212.006,E2 -8212.006} C_VEL
LIN {X 0,Y 462.696,Z 274.061,A -85,B 0,C 180,E1 -8213.733,E2 -8213.733} C_VEL
LIN {X 0,Y 462.994,Z 241.581,A -85,B 0,C 180,E1 -8214.258,E2 -8214.258} C_VEL
LIN {X 0,Y 459.245,Z 225.967,A -85,B 0,C 180,E1 -8214.734,E2 -8214.734} C_VEL
LIN {X 0,Y 456.827,Z 219.965,A -85,B 0,C 180,E1 -8214.987,E2 -8214.987} C_VEL
LIN {X 0,Y 454.024,Z 207.589,A -85,B 0,C 180,E1 -8217.419,E2 -8217.419} C_VEL
LIN {X 0,Y 453.552,Z 205.618,A -85,B 0,C 180,E1 -8217.87,E2 -8217.87} C_VEL
LIN {X 0,Y 453.465,Z 205.629,A -85,B 0,C 180,E1 -8221.525,E2 -8221.525} C_VEL
LIN {X 0,Y 453.486,Z 205.622,A -85,B 0,C 180,E1 -8224.777,E2 -8224.777} C_VEL
LIN {X 0,Y 453.47,Z 205.624,A -85,B 0,C 180,E1 -8228.31,E2 -8228.31} C_VEL
LIN {X 0,Y 453.491,Z 205.617,A -85,B 0,C 180,E1 -8230.608,E2 -8230.608} C_VEL
LIN {X 0,Y 453.46,Z 205.628,A -85,B 0,C 180,E1 -8233.245,E2 -8233.245} C_VEL
LIN {X 0,Y 453.461,Z 205.623,A -85,B 0,C 180,E1 -8235.778,E2 -8235.778} C_VEL
LIN {X 0,Y 453.511,Z 205.622,A -85,B 0,C 180,E1 -8239.405,E2 -8239.405} C_VEL
LIN {X 0,Y 453.47,Z 205.612,A -85,B 0,C 180,E1 -8242.222,E2 -8242.222} C_VEL
LIN {X 0,Y 453.483,Z 205.626,A -85,B 0,C 180,E1 -8245.222,E2 -8245.222} C_VEL
LIN {X 0,Y 453.462,Z 205.611,A -85,B 0,C 180,E1 -8248.474,E2 -8248.474} C_VEL
LIN {X 0,Y 453.507,Z 205.621,A -85,B 0,C 180,E1 -8251.288,E2 -8251.288} C_VEL
LIN {X 0,Y 453.517,Z 205.612,A -85,B 0,C 180,E1 -8254.284,E2 -8254.284} C_VEL
LIN {X 0,Y 453.471,Z 205.621,A -85,B 0,C 180,E1 -8257.204,E2 -8257.204} C_VEL
LIN {X 0,Y 453.497,Z 205.617,A -85,B 0,C 180,E1 -8260.066,E2 -8260.066} C_VEL
LIN {X 0,Y 453.499,Z 205.621,A -85,B 0,C 180,E1 -8262.875,E2 -8262.875} C_VEL
LIN {X 0,Y 453.505,Z 205.611,A -85,B 0,C 180,E1 -8265.643,E2 -8265.643} C_VEL
LIN {X 0,Y 453.553,Z 205.613,A -85,B 0,C 180,E1 -8268.379,E2 -8268.379} C_VEL
LIN {X 0,Y 453.643,Z 205.599,A -85,B 0,C 180,E1 -8271.985,E2 -8271.985} C_VEL
LIN {X 0,Y 453.662,Z 205.597,A -85,B 0,C 180,E1 -8274.667,E2 -8274.667} C_VEL
LIN {X 0,Y 453.756,Z 205.585,A -85,B 0,C 180,E1 -8277.337,E2 -8277.337} C_VEL
LIN {X 0,Y 453.814,Z 205.573,A -85,B 0,C 180,E1 -8280,E2 -8280} C_VEL
LIN {X 0,Y 453.756,Z 205.588,A -85,B 0,C 180,E1 -8282.663,E2 -8282.663} C_VEL
LIN {X 0,Y 453.668,Z 205.599,A -85,B 0,C 180,E1 -8286.225,E2 -8286.225} C_VEL
LIN {X 0,Y 453.584,Z 205.608,A -85,B 0,C 180,E1 -8288.913,E2 -8288.913} C_VEL
LIN {X 0,Y 453.554,Z 205.612,A -85,B 0,C 180,E1 -8292.529,E2 -8292.529} C_VEL
LIN {X 0,Y 453.548,Z 205.617,A -85,B 0,C 180,E1 -8296.196,E2 -8296.196} C_VEL
LIN {X 0,Y 453.512,Z 205.618,A -85,B 0,C 180,E1 -8299.041,E2 -8299.041} C_VEL
LIN {X 0,Y 453.468,Z 205.62,A -85,B 0,C 180,E1 -8301.836,E2 -8301.836} C_VEL
LIN {X 0,Y 453.506,Z 205.616,A -85,B 0,C 180,E1 -8304.735,E2 -8304.735} C_VEL
LIN {X 0,Y 453.531,Z 205.618,A -85,B 0,C 180,E1 -8307.962,E2 -8307.962} C_VEL
LIN {X 0,Y 453.476,Z 205.622,A -85,B 0,C 180,E1 -8310.759,E2 -8310.759} C_VEL
LIN {X 0,Y 453.471,Z 205.622,A -85,B 0,C 180,E1 -8313.913,E2 -8313.913} C_VEL
LIN {X 0,Y 453.447,Z 205.623,A -85,B 0,C 180,E1 -8317.19,E2 -8317.19} C_VEL
LIN {X 0,Y 453.499,Z 205.615,A -85,B 0,C 180,E1 -8319.449,E2 -8319.449} C_VEL
LIN {X 0,Y 453.457,Z 205.623,A -85,B 0,C 180,E1 -8322.996,E2 -8322.996} C_VEL
LIN {X 0,Y 453.461,Z 205.627,A -85,B 0,C 180,E1 -8325.78,E2 -8325.78} C_VEL
LIN {X 0,Y 453.512,Z 205.617,A -85,B 0,C 180,E1 -8329.406,E2 -8329.406} C_VEL
LIN {X 0,Y 453.472,Z 205.617,A -85,B 0,C 180,E1 -8332.224,E2 -8332.224} C_VEL
LIN {X 0,Y 453.485,Z 205.622,A -85,B 0,C 180,E1 -8335.223,E2 -8335.223} C_VEL
LIN {X 0,Y 453.463,Z 205.624,A -85,B 0,C 180,E1 -8338.475,E2 -8338.475} C_VEL
LIN {X 0,Y 453.529,Z 205.775,A -85,B 0,C 180,E1 -8338.938,E2 -8338.938} C_VEL
LIN {X 0,Y 457.142,Z 220.317,A -85,B 0,C 180,E1 -8341.538,E2 -8341.538} C_VEL
LIN {X 0,Y 458.606,Z 227.258,A -85,B 0,C 180,E1 -8342.727,E2 -8342.727} C_VEL
LIN {X 0,Y 457.62,Z 242.784,A -85,B 0,C 180,E1 -8345.099,E2 -8345.099} C_VEL
LIN {X 0,Y 462.809,Z 269.146,A -85,B 0,C 180,E1 -8345.838,E2 -8345.838} C_VEL
LIN {X 0,Y 461.253,Z 391.882,A -85,B 0,C 180,E1 -8347.787,E2 -8347.787} C_VEL
LIN {X 0,Y 460.897,Z 412.094,A -85,B 0,C 180,E1 -8348.152,E2 -8348.152} C_VEL
LIN {X 0,Y 460.26,Z 427.655,A -85,B 0,C 180,E1 -8348.608,E2 -8348.608} C_VEL
LIN {X 0,Y 459.599,Z 441.884,A -85,B 0,C 180,E1 -8349.2,E2 -8349.2} C_VEL
LIN {X 0,Y 458.703,Z 455.85,A -85,B 0,C 180,E1 -8349.952,E2 -8349.952} C_VEL
LIN {X 0,Y 457.837,Z 469.062,A -85,B 0,C 180,E1 -8350.846,E2 -8350.846} C_VEL
LIN {X 0,Y 456.771,Z 482.514,A -85,B 0,C 180,E1 -8351.962,E2 -8351.962} C_VEL
LIN {X 0,Y 455.874,Z 494.771,A -85,B 0,C 180,E1 -8353.199,E2 -8353.199} C_VEL
LIN {X 0,Y 454.961,Z 505.964,A -85,B 0,C 180,E1 -8354.546,E2 -8354.546} C_VEL
LIN {X 0,Y 454.145,Z 516.828,A -85,B 0,C 180,E1 -8356.122,E2 -8356.122} C_VEL
LIN {X 0,Y 453.555,Z 525.593,A -85,B 0,C 180,E1 -8357.643,E2 -8357.643} C_VEL
LIN {X 0,Y 453.168,Z 533.39,A -85,B 0,C 180,E1 -8359.275,E2 -8359.275} C_VEL
LIN {X 0,Y 452.781,Z 540.398,A -85,B 0,C 180,E1 -8361.071,E2 -8361.071} C_VEL
LIN {X 0,Y 452.645,Z 545.911,A -85,B 0,C 180,E1 -8362.865,E2 -8362.865} C_VEL
LIN {X 0,Y 452.509,Z 550.078,A -85,B 0,C 180,E1 -8364.653,E2 -8364.653} C_VEL
LIN {X 0,Y 452.427,Z 553,A -85,B 0,C 180,E1 -8366.438,E2 -8366.438} C_VEL
LIN {X 0,Y 452.433,Z 554.743,A -85,B 0,C 180,E1 -8368.22,E2 -8368.22} C_VEL
LIN {X 0,Y 452.431,Z 555.341,A -85,B 0,C 180,E1 -8370,E2 -8370} C_VEL
LIN {X 0,Y 452.433,Z 554.74,A -85,B 0,C 180,E1 -8371.78,E2 -8371.78} C_VEL
LIN {X 0,Y 452.427,Z 552.993,A -85,B 0,C 180,E1 -8373.562,E2 -8373.562} C_VEL
LIN {X 0,Y 452.516,Z 550.073,A -85,B 0,C 180,E1 -8375.347,E2 -8375.347} C_VEL
LIN {X 0,Y 452.647,Z 545.911,A -85,B 0,C 180,E1 -8377.135,E2 -8377.135} C_VEL
LIN {X 0,Y 452.781,Z 540.393,A -85,B 0,C 180,E1 -8378.929,E2 -8378.929} C_VEL
LIN {X 0,Y 453.167,Z 533.376,A -85,B 0,C 180,E1 -8380.725,E2 -8380.725} C_VEL
LIN {X 0,Y 453.546,Z 525.607,A -85,B 0,C 180,E1 -8382.352,E2 -8382.352} C_VEL
LIN {X 0,Y 454.144,Z 516.816,A -85,B 0,C 180,E1 -8383.878,E2 -8383.878} C_VEL
LIN {X 0,Y 454.954,Z 505.946,A -85,B 0,C 180,E1 -8385.454,E2 -8385.454} C_VEL
LIN {X 0,Y 455.856,Z 494.755,A -85,B 0,C 180,E1 -8386.802,E2 -8386.802} C_VEL
LIN {X 0,Y 456.823,Z 482.498,A -85,B 0,C 180,E1 -8388.035,E2 -8388.035} C_VEL
LIN {X 0,Y 457.885,Z 469.027,A -85,B 0,C 180,E1 -8389.152,E2 -8389.152} C_VEL
LIN {X 0,Y 458.72,Z 455.797,A -85,B 0,C 180,E1 -8390.047,E2 -8390.047} C_VEL
LIN {X 0,Y 459.599,Z 441.801,A -85,B 0,C 180,E1 -8390.801,E2 -8390.801} C_VEL
LIN {X 0,Y 460.316,Z 427.095,A -85,B 0,C 180,E1 -8391.409,E2 -8391.409} C_VEL
LIN {X 0,Y 460.865,Z 411.973,A -85,B 0,C 180,E1 -8391.85,E2 -8391.85} C_VEL
LIN {X 0,Y 461.277,Z 389.885,A -85,B 0,C 180,E1 -8392.241,E2 -8392.241} C_VEL
LIN {X 0,Y 462.818,Z 269.047,A -85,B 0,C 180,E1 -8394.159,E2 -8394.159} C_VEL
LIN {X 0,Y 457.658,Z 242.617,A -85,B 0,C 180,E1 -8394.919,E2 -8394.919} C_VEL
LIN {X 0,Y 458.581,Z 227.267,A -85,B 0,C 180,E1 -8397.267,E2 -8397.267} C_VEL
LIN {X 0,Y 455.968,Z 215.452,A -85,B 0,C 180,E1 -8399.312,E2 -8399.312} C_VEL
LIN {X 0,Y 453.512,Z 205.614,A -85,B 0,C 180,E1 -8401.124,E2 -8401.124} C_VEL
LIN {X 0,Y 453.475,Z 205.615,A -85,B 0,C 180,E1 -8403.912,E2 -8403.912} C_VEL
LIN {X 0,Y 453.467,Z 205.623,A -85,B 0,C 180,E1 -8407.187,E2 -8407.187} C_VEL
LIN {X 0,Y 453.524,Z 205.617,A -85,B 0,C 180,E1 -8409.445,E2 -8409.445} C_VEL
LIN {X 0,Y 453.474,Z 205.625,A -85,B 0,C 180,E1 -8411.935,E2 -8411.935} C_VEL
LIN {X 0,Y 453.482,Z 205.619,A -85,B 0,C 180,E1 -8415.47,E2 -8415.47} C_VEL
LIN {X 0,Y 453.476,Z 205.622,A -85,B 0,C 180,E1 -8418.209,E2 -8418.209} C_VEL
LIN {X 0,Y 453.52,Z 205.612,A -85,B 0,C 180,E1 -8420.788,E2 -8420.788} C_VEL
LIN {X 0,Y 453.45,Z 205.624,A -85,B 0,C 180,E1 -8423.917,E2 -8423.917} C_VEL
LIN {X 0,Y 453.476,Z 205.616,A -85,B 0,C 180,E1 -8427.151,E2 -8427.151} C_VEL
LIN {X 0,Y 453.507,Z 205.616,A -85,B 0,C 180,E1 -8430.271,E2 -8430.271} C_VEL
LIN {X 0,Y 453.501,Z 205.617,A -85,B 0,C 180,E1 -8433.294,E2 -8433.294} C_VEL
LIN {X 0,Y 453.495,Z 205.615,A -85,B 0,C 180,E1 -8436.238,E2 -8436.238} C_VEL
LIN {X 0,Y 453.474,Z 205.608,A -85,B 0,C 180,E1 -8439.117,E2 -8439.117} C_VEL
LIN {X 0,Y 453.503,Z 205.619,A -85,B 0,C 180,E1 -8441.944,E2 -8441.944} C_VEL
LIN {X 0,Y 453.531,Z 205.612,A -85,B 0,C 180,E1 -8444.726,E2 -8444.726} C_VEL
LIN {X 0,Y 453.552,Z 205.609,A -85,B 0,C 180,E1 -8448.379,E2 -8448.379} C_VEL
LIN {X 0,Y 453.643,Z 205.599,A -85,B 0,C 180,E1 -8451.985,E2 -8451.985} C_VEL
LIN {X 0,Y 453.663,Z 205.596,A -85,B 0,C 180,E1 -8454.667,E2 -8454.667} C_VEL
LIN {X 0,Y 453.757,Z 205.589,A -85,B 0,C 180,E1 -8457.337,E2 -8457.337} C_VEL
LIN {X 0,Y 453.814,Z 205.575,A -85,B 0,C 180,E1 -8460,E2 -8460} C_VEL
LIN {X 0,Y 453.757,Z 205.585,A -85,B 0,C 180,E1 -8462.663,E2 -8462.663} C_VEL
LIN {X 0,Y 453.671,Z 205.595,A -85,B 0,C 180,E1 -8466.225,E2 -8466.225} C_VEL
LIN {X 0,Y 453.584,Z 205.606,A -85,B 0,C 180,E1 -8468.914,E2 -8468.914} C_VEL
LIN {X 0,Y 453.555,Z 205.608,A -85,B 0,C 180,E1 -8472.529,E2 -8472.529} C_VEL
LIN {X 0,Y 453.536,Z 205.61,A -85,B 0,C 180,E1 -8476.196,E2 -8476.196} C_VEL
LIN {X 0,Y 453.512,Z 205.622,A -85,B 0,C 180,E1 -8479.041,E2 -8479.041} C_VEL
LIN {X 0,Y 453.468,Z 205.621,A -85,B 0,C 180,E1 -8481.837,E2 -8481.837} C_VEL
LIN {X 0,Y 453.506,Z 205.615,A -85,B 0,C 180,E1 -8484.735,E2 -8484.735} C_VEL
LIN {X 0,Y 453.532,Z 205.61,A -85,B 0,C 180,E1 -8487.962,E2 -8487.962} C_VEL
LIN {X 0,Y 453.477,Z 205.623,A -85,B 0,C 180,E1 -8490.76,E2 -8490.76} C_VEL
LIN {X 0,Y 453.472,Z 205.617,A -85,B 0,C 180,E1 -8493.913,E2 -8493.913} C_VEL
LIN {X 0,Y 453.465,Z 205.624,A -85,B 0,C 180,E1 -8497.189,E2 -8497.189} C_VEL
LIN {X 0,Y 453.484,Z 205.617,A -85,B 0,C 180,E1 -8499.45,E2 -8499.45} C_VEL
LIN {X 0,Y 453.471,Z 205.617,A -85,B 0,C 180,E1 -8501.936,E2 -8501.936} C_VEL
LIN {X 0,Y 453.487,Z 205.619,A -85,B 0,C 180,E1 -8505.471,E2 -8505.471} C_VEL
LIN {X 0,Y 453.478,Z 205.622,A -85,B 0,C 180,E1 -8508.21,E2 -8508.21} C_VEL
LIN {X 0,Y 453.512,Z 205.616,A -85,B 0,C 180,E1 -8510.791,E2 -8510.791} C_VEL
LIN {X 0,Y 453.451,Z 205.623,A -85,B 0,C 180,E1 -8513.918,E2 -8513.918} C_VEL
LIN {X 0,Y 453.481,Z 205.623,A -85,B 0,C 180,E1 -8517.152,E2 -8517.152} C_VEL
LIN {X 0,Y 453.474,Z 205.625,A -85,B 0,C 180,E1 -8520.269,E2 -8520.269} C_VEL
LIN {X 0,Y 453.574,Z 205.724,A -85,B 0,C 180,E1 -8522.301,E2 -8522.301} C_VEL
LIN {X 0,Y 456.802,Z 219.993,A -85,B 0,C 180,E1 -8525.109,E2 -8525.109} C_VEL
LIN {X 0,Y 459.857,Z 228.046,A -85,B 0,C 180,E1 -8525.431,E2 -8525.431} C_VEL
LIN {X 0,Y 463.089,Z 242.727,A -85,B 0,C 180,E1 -8525.861,E2 -8525.861} C_VEL
LIN {X 0,Y 461.855,Z 340.549,A -85,B 0,C 180,E1 -8527.418,E2 -8527.418} C_VEL
LIN {X 0,Y 461.116,Z 346.402,A -85,B 0,C 180,E1 -8527.476,E2 -8527.476} C_VEL
LIN {X 0,Y 455.499,Z 365.44,A -85,B 0,C 180,E1 -8527.499,E2 -8527.499} C_VEL
LIN {X 0,Y 454.894,Z 371.284,A -85,B 0,C 180,E1 -8527.565,E2 -8527.565} C_VEL
LIN {X 0,Y 454.515,Z 389.092,A -85,B 0,C 180,E1 -8527.904,E2 -8527.904} C_VEL
LIN {X 0,Y 453.974,Z 404.749,A -85,B 0,C 180,E1 -8528.39,E2 -8528.39} C_VEL
LIN {X 0,Y 453.302,Z 419.081,A -85,B 0,C 180,E1 -8529.015,E2 -8529.015} C_VEL
LIN {X 0,Y 452.419,Z 432.687,A -85,B 0,C 180,E1 -8529.78,E2 -8529.78} C_VEL
LIN {X 0,Y 451.524,Z 445.615,A -85,B 0,C 180,E1 -8530.686,E2 -8530.686} C_VEL
LIN {X 0,Y 450.604,Z 457.653,A -85,B 0,C 180,E1 -8531.707,E2 -8531.707} C_VEL
LIN {X 0,Y 449.582,Z 469.868,A -85,B 0,C 180,E1 -8532.956,E2 -8532.956} C_VEL
LIN {X 0,Y 448.644,Z 480.99,A -85,B 0,C 180,E1 -8534.323,E2 -8534.323} C_VEL
LIN {X 0,Y 447.722,Z 491.792,A -85,B 0,C 180,E1 -8535.919,E2 -8535.919} C_VEL
LIN {X 0,Y 446.985,Z 500.754,A -85,B 0,C 180,E1 -8537.515,E2 -8537.515} C_VEL
LIN {X 0,Y 446.451,Z 508.178,A -85,B 0,C 180,E1 -8539.111,E2 -8539.111} C_VEL
LIN {X 0,Y 446.002,Z 515.118,A -85,B 0,C 180,E1 -8540.934,E2 -8540.934} C_VEL
LIN {X 0,Y 445.719,Z 520.572,A -85,B 0,C 180,E1 -8542.753,E2 -8542.753} C_VEL
LIN {X 0,Y 445.579,Z 524.689,A -85,B 0,C 180,E1 -8544.57,E2 -8544.57} C_VEL
LIN {X 0,Y 445.441,Z 527.585,A -85,B 0,C 180,E1 -8546.382,E2 -8546.382} C_VEL
LIN {X 0,Y 445.377,Z 529.328,A -85,B 0,C 180,E1 -8548.191,E2 -8548.191} C_VEL
LIN {X 0,Y 445.34,Z 529.939,A -85,B 0,C 180,E1 -8550,E2 -8550} C_VEL
LIN {X 0,Y 445.377,Z 529.379,A -85,B 0,C 180,E1 -8551.808,E2 -8551.808} C_VEL
LIN {X 0,Y 445.441,Z 527.703,A -85,B 0,C 180,E1 -8553.618,E2 -8553.618} C_VEL
LIN {X 0,Y 445.57,Z 524.871,A -85,B 0,C 180,E1 -8555.43,E2 -8555.43} C_VEL
LIN {X 0,Y 445.714,Z 520.818,A -85,B 0,C 180,E1 -8557.247,E2 -8557.247} C_VEL
LIN {X 0,Y 445.993,Z 515.441,A -85,B 0,C 180,E1 -8559.066,E2 -8559.066} C_VEL
LIN {X 0,Y 446.428,Z 508.588,A -85,B 0,C 180,E1 -8560.889,E2 -8560.889} C_VEL
LIN {X 0,Y 446.968,Z 501.216,A -85,B 0,C 180,E1 -8562.486,E2 -8562.486} C_VEL
LIN {X 0,Y 447.683,Z 492.332,A -85,B 0,C 180,E1 -8564.083,E2 -8564.083} C_VEL
LIN {X 0,Y 448.435,Z 483.273,A -85,B 0,C 180,E1 -8565.451,E2 -8565.451} C_VEL
LIN {X 0,Y 449.328,Z 472.584,A -85,B 0,C 180,E1 -8566.819,E2 -8566.819} C_VEL
LIN {X 0,Y 450.346,Z 461.012,A -85,B 0,C 180,E1 -8568.058,E2 -8568.058} C_VEL
LIN {X 0,Y 451.38,Z 448.16,A -85,B 0,C 180,E1 -8569.203,E2 -8569.203} C_VEL
LIN {X 0,Y 452.336,Z 434.089,A -85,B 0,C 180,E1 -8570.224,E2 -8570.224} C_VEL
LIN {X 0,Y 453.305,Z 419.442,A -85,B 0,C 180,E1 -8571.059,E2 -8571.059} C_VEL
LIN {X 0,Y 453.959,Z 404.357,A -85,B 0,C 180,E1 -8571.72,E2 -8571.72} C_VEL
LIN {X 0,Y 454.525,Z 388.673,A -85,B 0,C 180,E1 -8572.201,E2 -8572.201} C_VEL
LIN {X 0,Y 454.934,Z 368.834,A -85,B 0,C 180,E1 -8572.568,E2 -8572.568} C_VEL
LIN {X 0,Y 456.304,Z 267.611,A -85,B 0,C 180,E1 -8574.198,E2 -8574.198} C_VEL
LIN {X 0,Y 456.51,Z 242.721,A -85,B 0,C 180,E1 -8574.608,E2 -8574.608} C_VEL
LIN {X 0,Y 453.1,Z 228.57,A -85,B 0,C 180,E1 -8575.05,E2 -8575.05} C_VEL
LIN {X 0,Y 449.651,Z 220.117,A -85,B 0,C 180,E1 -8575.425,E2 -8575.425} C_VEL
LIN {X 0,Y 447.138,Z 209.126,A -85,B 0,C 180,E1 -8577.624,E2 -8577.624} C_VEL
LIN {X 0,Y 446.484,Z 206.497,A -85,B 0,C 180,E1 -8578.178,E2 -8578.178} C_VEL
LIN {X 0,Y 446.418,Z 206.507,A -85,B 0,C 180,E1 -8581.774,E2 -8581.774} C_VEL
LIN {X 0,Y 446.428,Z 206.501,A -85,B 0,C 180,E1 -8584.522,E2 -8584.522} C_VEL
LIN {X 0,Y 446.428,Z 206.503,A -85,B 0,C 180,E1 -8588.081,E2 -8588.081} C_VEL
LIN {X 0,Y 446.425,Z 206.5,A -85,B 0,C 180,E1 -8590.917,E2 -8590.917} C_VEL
LIN {X 0,Y 446.419,Z 206.5,A -85,B 0,C 180,E1 -8593.842,E2 -8593.842} C_VEL
LIN {X 0,Y 446.395,Z 206.501,A -85,B 0,C 180,E1 -8596.403,E2 -8596.403} C_VEL
LIN {X 0,Y 446.463,Z 206.495,A -85,B 0,C 180,E1 -8599.804,E2 -8599.804} C_VEL
LIN {X 0,Y 446.426,Z 206.489,A -85,B 0,C 180,E1 -8602.123,E2 -8602.123} C_VEL
LIN {X 0,Y 446.424,Z 206.501,A -85,B 0,C 180,E1 -8605.476,E2 -8605.476} C_VEL
LIN {X 0,Y 446.413,Z 206.488,A -85,B 0,C 180,E1 -8608.699,E2 -8608.699} C_VEL
LIN {X 0,Y 446.477,Z 206.492,A -85,B 0,C 180,E1 -8611.821,E2 -8611.821} C_VEL
LIN {X 0,Y 446.45,Z 206.497,A -85,B 0,C 180,E1 -8614.847,E2 -8614.847} C_VEL
LIN {X 0,Y 446.44,Z 206.494,A -85,B 0,C 180,E1 -8618.245,E2 -8618.245} C_VEL
LIN {X 0,Y 446.449,Z 206.492,A -85,B 0,C 180,E1 -8621.649,E2 -8621.649} C_VEL
LIN {X 0,Y 446.499,Z 206.492,A -85,B 0,C 180,E1 -8624.479,E2 -8624.479} C_VEL
LIN {X 0,Y 446.51,Z 206.489,A -85,B 0,C 180,E1 -8628.193,E2 -8628.193} C_VEL
LIN {X 0,Y 446.591,Z 206.477,A -85,B 0,C 180,E1 -8631.858,E2 -8631.858} C_VEL
LIN {X 0,Y 446.637,Z 206.472,A -85,B 0,C 180,E1 -8634.582,E2 -8634.582} C_VEL
LIN {X 0,Y 446.7,Z 206.465,A -85,B 0,C 180,E1 -8637.295,E2 -8637.295} C_VEL
LIN {X 0,Y 446.785,Z 206.449,A -85,B 0,C 180,E1 -8640,E2 -8640} C_VEL
LIN {X 0,Y 446.7,Z 206.466,A -85,B 0,C 180,E1 -8642.705,E2 -8642.705} C_VEL
LIN {X 0,Y 446.637,Z 206.476,A -85,B 0,C 180,E1 -8646.324,E2 -8646.324} C_VEL
LIN {X 0,Y 446.53,Z 206.486,A -85,B 0,C 180,E1 -8649.055,E2 -8649.055} C_VEL
LIN {X 0,Y 446.513,Z 206.488,A -85,B 0,C 180,E1 -8652.73,E2 -8652.73} C_VEL
LIN {X 0,Y 446.51,Z 206.494,A -85,B 0,C 180,E1 -8656.238,E2 -8656.238} C_VEL
LIN {X 0,Y 446.461,Z 206.495,A -85,B 0,C 180,E1 -8659.303,E2 -8659.303} C_VEL
LIN {X 0,Y 446.41,Z 206.502,A -85,B 0,C 180,E1 -8662.2,E2 -8662.2} C_VEL
LIN {X 0,Y 446.449,Z 206.492,A -85,B 0,C 180,E1 -8665.153,E2 -8665.153} C_VEL
LIN {X 0,Y 446.477,Z 206.498,A -85,B 0,C 180,E1 -8668.179,E2 -8668.179} C_VEL
LIN {X 0,Y 446.412,Z 206.5,A -85,B 0,C 180,E1 -8671.301,E2 -8671.301} C_VEL
LIN {X 0,Y 446.424,Z 206.502,A -85,B 0,C 180,E1 -8674.523,E2 -8674.523} C_VEL
LIN {X 0,Y 446.409,Z 206.506,A -85,B 0,C 180,E1 -8678.08,E2 -8678.08} C_VEL
LIN {X 0,Y 446.421,Z 206.489,A -85,B 0,C 180,E1 -8680.918,E2 -8680.918} C_VEL
LIN {X 0,Y 446.396,Z 206.507,A -85,B 0,C 180,E1 -8683.846,E2 -8683.846} C_VEL
LIN {X 0,Y 446.394,Z 206.505,A -85,B 0,C 180,E1 -8686.404,E2 -8686.404} C_VEL
LIN {X 0,Y 446.463,Z 206.497,A -85,B 0,C 180,E1 -8689.805,E2 -8689.805} C_VEL
LIN {X 0,Y 446.427,Z 206.495,A -85,B 0,C 180,E1 -8692.124,E2 -8692.124} C_VEL
LIN {X 0,Y 446.427,Z 206.503,A -85,B 0,C 180,E1 -8695.478,E2 -8695.478} C_VEL
LIN {X 0,Y 446.446,Z 206.661,A -85,B 0,C 180,E1 -8698.572,E2 -8698.572} C_VEL
LIN {X 0,Y 450.117,Z 221.271,A -85,B 0,C 180,E1 -8701.24,E2 -8701.24} C_VEL
LIN {X 0,Y 451.755,Z 229.487,A -85,B 0,C 180,E1 -8702.667,E2 -8702.667} C_VEL
LIN {X 0,Y 450.884,Z 242.548,A -85,B 0,C 180,E1 -8704.696,E2 -8704.696} C_VEL
LIN {X 0,Y 456.372,Z 271.044,A -85,B 0,C 180,E1 -8705.511,E2 -8705.511} C_VEL
LIN {X 0,Y 454.412,Z 408.31,A -85,B 0,C 180,E1 -8707.734,E2 -8707.734} C_VEL
LIN {X 0,Y 453.889,Z 423.861,A -85,B 0,C 180,E1 -8708.155,E2 -8708.155} C_VEL
LIN {X 0,Y 453.11,Z 438.678,A -85,B 0,C 180,E1 -8708.736,E2 -8708.736} C_VEL
LIN {X 0,Y 452.265,Z 451.848,A -85,B 0,C 180,E1 -8709.416,E2 -8709.416} C_VEL
LIN {X 0,Y 451.281,Z 465.758,A -85,B 0,C 180,E1 -8710.32,E2 -8710.32} C_VEL
LIN {X 0,Y 450.275,Z 478.505,A -85,B 0,C 180,E1 -8711.339,E2 -8711.339} C_VEL
LIN {X 0,Y 449.359,Z 490.331,A -85,B 0,C 180,E1 -8712.479,E2 -8712.479} C_VEL
LIN {X 0,Y 448.365,Z 502.2,A -85,B 0,C 180,E1 -8713.846,E2 -8713.846} C_VEL
LIN {X 0,Y 447.557,Z 512.195,A -85,B 0,C 180,E1 -8715.216,E2 -8715.216} C_VEL
LIN {X 0,Y 446.767,Z 521.975,A -85,B 0,C 180,E1 -8716.815,E2 -8716.815} C_VEL
LIN {X 0,Y 446.293,Z 530.142,A -85,B 0,C 180,E1 -8718.418,E2 -8718.418} C_VEL
LIN {X 0,Y 445.824,Z 536.89,A -85,B 0,C 180,E1 -8720.014,E2 -8720.014} C_VEL
LIN {X 0,Y 445.606,Z 543.128,A -85,B 0,C 180,E1 -8721.84,E2 -8721.84} C_VEL
LIN {X 0,Y 445.451,Z 548.056,A -85,B 0,C 180,E1 -8723.703,E2 -8723.703} C_VEL
LIN {X 0,Y 445.36,Z 551.489,A -85,B 0,C 180,E1 -8725.475,E2 -8725.475} C_VEL
LIN {X 0,Y 445.418,Z 553.817,A -85,B 0,C 180,E1 -8727.287,E2 -8727.287} C_VEL
LIN {X 0,Y 445.336,Z 554.986,A -85,B 0,C 180,E1 -8729.096,E2 -8729.096} C_VEL
LIN {X 0,Y 445.336,Z 554.985,A -85,B 0,C 180,E1 -8730.904,E2 -8730.904} C_VEL
LIN {X 0,Y 445.418,Z 553.812,A -85,B 0,C 180,E1 -8732.713,E2 -8732.713} C_VEL
LIN {X 0,Y 445.361,Z 551.481,A -85,B 0,C 180,E1 -8734.525,E2 -8734.525} C_VEL
LIN {X 0,Y 445.488,Z 547.951,A -85,B 0,C 180,E1 -8736.34,E2 -8736.34} C_VEL
LIN {X 0,Y 445.606,Z 543.126,A -85,B 0,C 180,E1 -8738.16,E2 -8738.16} C_VEL
LIN {X 0,Y 445.824,Z 536.877,A -85,B 0,C 180,E1 -8739.986,E2 -8739.986} C_VEL
LIN {X 0,Y 446.294,Z 530.125,A -85,B 0,C 180,E1 -8741.582,E2 -8741.582} C_VEL
LIN {X 0,Y 446.766,Z 521.96,A -85,B 0,C 180,E1 -8743.185,E2 -8743.185} C_VEL
LIN {X 0,Y 447.564,Z 512.178,A -85,B 0,C 180,E1 -8744.783,E2 -8744.783} C_VEL
LIN {X 0,Y 448.382,Z 502.179,A -85,B 0,C 180,E1 -8746.153,E2 -8746.153} C_VEL
LIN {X 0,Y 449.354,Z 490.523,A -85,B 0,C 180,E1 -8747.498,E2 -8747.498} C_VEL
LIN {X 0,Y 450.278,Z 478.477,A -85,B 0,C 180,E1 -8748.66,E2 -8748.66} C_VEL
LIN {X 0,Y 451.291,Z 465.708,A -85,B 0,C 180,E1 -8749.68,E2 -8749.68} C_VEL
LIN {X 0,Y 452.259,Z 451.781,A -85,B 0,C 180,E1 -8750.584,E2 -8750.584} C_VEL
LIN {X 0,Y 453.186,Z 437.369,A -85,B 0,C 180,E1 -8751.317,E2 -8751.317} C_VEL
LIN {X 0,Y 453.868,Z 421.924,A -85,B 0,C 180,E1 -8751.905,E2 -8751.905} C_VEL
LIN {X 0,Y 454.458,Z 406.608,A -85,B 0,C 180,E1 -8752.294,E2 -8752.294} C_VEL
LIN {X 0,Y 456.409,Z 271.112,A -85,B 0,C 180,E1 -8754.482,E2 -8754.482} C_VEL
LIN {X 0,Y 450.908,Z 242.46,A -85,B 0,C 180,E1 -8755.31,E2 -8755.31} C_VEL
LIN {X 0,Y 451.688,Z 228.327,A -85,B 0,C 180,E1 -8757.516,E2 -8757.516} C_VEL
LIN {X 0,Y 448.704,Z 215.321,A -85,B 0,C 180,E1 -8759.82,E2 -8759.82} C_VEL
LIN {X 0,Y 446.424,Z 206.496,A -85,B 0,C 180,E1 -8761.474,E2 -8761.474} C_VEL
LIN {X 0,Y 446.427,Z 206.498,A -85,B 0,C 180,E1 -8764.522,E2 -8764.522} C_VEL
LIN {X 0,Y 446.432,Z 206.504,A -85,B 0,C 180,E1 -8768.082,E2 -8768.082} C_VEL
LIN {X 0,Y 446.439,Z 206.497,A -85,B 0,C 180,E1 -8770.919,E2 -8770.919} C_VEL
LIN {X 0,Y 446.396,Z 206.506,A -85,B 0,C 180,E1 -8773.845,E2 -8773.845} C_VEL
LIN {X 0,Y 446.394,Z 206.502,A -85,B 0,C 180,E1 -8776.403,E2 -8776.403} C_VEL
LIN {X 0,Y 446.461,Z 206.495,A -85,B 0,C 180,E1 -8779.804,E2 -8779.804} C_VEL
LIN {X 0,Y 446.425,Z 206.499,A -85,B 0,C 180,E1 -8782.123,E2 -8782.123} C_VEL
LIN {X 0,Y 446.424,Z 206.497,A -85,B 0,C 180,E1 -8785.477,E2 -8785.477} C_VEL
LIN {X 0,Y 446.412,Z 206.498,A -85,B 0,C 180,E1 -8788.699,E2 -8788.699} C_VEL
LIN {X 0,Y 446.477,Z 206.496,A -85,B 0,C 180,E1 -8791.821,E2 -8791.821} C_VEL
LIN {X 0,Y 446.449,Z 206.495,A -85,B 0,C 180,E1 -8794.847,E2 -8794.847} C_VEL
LIN {X 0,Y 446.44,Z 206.483,A -85,B 0,C 180,E1 -8798.245,E2 -8798.245} C_VEL
LIN {X 0,Y 446.449,Z 206.502,A -85,B 0,C 180,E1 -8801.649,E2 -8801.649} C_VEL
LIN {X 0,Y 446.499,Z 206.488,A -85,B 0,C 180,E1 -8804.48,E2 -8804.48} C_VEL
LIN {X 0,Y 446.51,Z 206.487,A -85,B 0,C 180,E1 -8808.193,E2 -8808.193} C_VEL
LIN {X 0,Y 446.591,Z 206.479,A -85,B 0,C 180,E1 -8811.858,E2 -8811.858} C_VEL
LIN {X 0,Y 446.637,Z 206.471,A -85,B 0,C 180,E1 -8814.583,E2 -8814.583} C_VEL
LIN {X 0,Y 446.701,Z 206.467,A -85,B 0,C 180,E1 -8817.295,E2 -8817.295} C_VEL
LIN {X 0,Y 446.785,Z 206.45,A -85,B 0,C 180,E1 -8820,E2 -8820} C_VEL
LIN {X 0,Y 446.701,Z 206.465,A -85,B 0,C 180,E1 -8822.705,E2 -8822.705} C_VEL
LIN {X 0,Y 446.64,Z 206.471,A -85,B 0,C 180,E1 -8826.324,E2 -8826.324} C_VEL
LIN {X 0,Y 446.53,Z 206.485,A -85,B 0,C 180,E1 -8829.056,E2 -8829.056} C_VEL
LIN {X 0,Y 446.515,Z 206.486,A -85,B 0,C 180,E1 -8832.73,E2 -8832.73} C_VEL
LIN {X 0,Y 446.488,Z 206.488,A -85,B 0,C 180,E1 -8836.228,E2 -8836.228} C_VEL
LIN {X 0,Y 446.461,Z 206.497,A -85,B 0,C 180,E1 -8839.304,E2 -8839.304} C_VEL
LIN {X 0,Y 446.41,Z 206.5,A -85,B 0,C 180,E1 -8842.2,E2 -8842.2} C_VEL
LIN {X 0,Y 446.45,Z 206.485,A -85,B 0,C 180,E1 -8845.153,E2 -8845.153} C_VEL
LIN {X 0,Y 446.478,Z 206.489,A -85,B 0,C 180,E1 -8848.179,E2 -8848.179} C_VEL
LIN {X 0,Y 446.413,Z 206.503,A -85,B 0,C 180,E1 -8851.301,E2 -8851.301} C_VEL
LIN {X 0,Y 446.424,Z 206.498,A -85,B 0,C 180,E1 -8854.524,E2 -8854.524} C_VEL
LIN {X 0,Y 446.425,Z 206.497,A -85,B 0,C 180,E1 -8858.082,E2 -8858.082} C_VEL
LIN {X 0,Y 446.422,Z 206.502,A -85,B 0,C 180,E1 -8860.918,E2 -8860.918} C_VEL
LIN {X 0,Y 446.419,Z 206.497,A -85,B 0,C 180,E1 -8863.844,E2 -8863.844} C_VEL
LIN {X 0,Y 446.417,Z 206.502,A -85,B 0,C 180,E1 -8866.401,E2 -8866.401} C_VEL
LIN {X 0,Y 446.448,Z 206.497,A -85,B 0,C 180,E1 -8869.804,E2 -8869.804} C_VEL
LIN {X 0,Y 446.406,Z 206.502,A -85,B 0,C 180,E1 -8872.122,E2 -8872.122} C_VEL
LIN {X 0,Y 446.426,Z 206.501,A -85,B 0,C 180,E1 -8875.478,E2 -8875.478} C_VEL
LIN {X 0,Y 446.415,Z 206.502,A -85,B 0,C 180,E1 -8878.7,E2 -8878.7} C_VEL
LIN {X 0,Y 446.501,Z 206.613,A -85,B 0,C 180,E1 -8881.954,E2 -8881.954} C_VEL
LIN {X 0,Y 449.486,Z 219.43,A -85,B 0,C 180,E1 -8884.534,E2 -8884.534} C_VEL
LIN {X 0,Y 449.771,Z 220.637,A -85,B 0,C 180,E1 -8884.708,E2 -8884.708} C_VEL
LIN {X 0,Y 453.726,Z 230.681,A -85,B 0,C 180,E1 -8885.118,E2 -8885.118} C_VEL
LIN {X 0,Y 456.626,Z 243.875,A -85,B 0,C 180,E1 -8885.513,E2 -8885.513} C_VEL
LIN {X 0,Y 455.14,Z 352.492,A -85,B 0,C 180,E1 -8887.263,E2 -8887.263} C_VEL
LIN {X 0,Y 454.894,Z 371.284,A -85,B 0,C 180,E1 -8887.565,E2 -8887.565} C_VEL
LIN {X 0,Y 454.268,Z 377.137,A -85,B 0,C 180,E1 -8887.63,E2 -8887.63} C_VEL
LIN {X 0,Y 448.89,Z 394.162,A -85,B 0,C 180,E1 -8887.742,E2 -8887.742} C_VEL
LIN {X 0,Y 447.706,Z 399.852,A -85,B 0,C 180,E1 -8887.871,E2 -8887.871} C_VEL
LIN {X 0,Y 447.559,Z 401.745,A -85,B 0,C 180,E1 -8887.936,E2 -8887.936} C_VEL
LIN {X 0,Y 446.879,Z 415.958,A -85,B 0,C 180,E1 -8888.521,E2 -8888.521} C_VEL
LIN {X 0,Y 446.033,Z 429.244,A -85,B 0,C 180,E1 -8889.236,E2 -8889.236} C_VEL
LIN {X 0,Y 445.086,Z 442.829,A -85,B 0,C 180,E1 -8890.155,E2 -8890.155} C_VEL
LIN {X 0,Y 444.035,Z 455.32,A -85,B 0,C 180,E1 -8891.187,E2 -8891.187} C_VEL
LIN {X 0,Y 443.137,Z 466.152,A -85,B 0,C 180,E1 -8892.26,E2 -8892.26} C_VEL
LIN {X 0,Y 442.076,Z 477.656,A -85,B 0,C 180,E1 -8893.61,E2 -8893.61} C_VEL
LIN {X 0,Y 441.234,Z 487.593,A -85,B 0,C 180,E1 -8895,E2 -8895} C_VEL
LIN {X 0,Y 440.43,Z 496.163,A -85,B 0,C 180,E1 -8896.411,E2 -8896.411} C_VEL
LIN {X 0,Y 439.815,Z 504.289,A -85,B 0,C 180,E1 -8898.011,E2 -8898.011} C_VEL
LIN {X 0,Y 439.187,Z 512.049,A -85,B 0,C 180,E1 -8899.862,E2 -8899.862} C_VEL
LIN {X 0,Y 438.813,Z 518.223,A -85,B 0,C 180,E1 -8901.713,E2 -8901.713} C_VEL
LIN {X 0,Y 438.593,Z 522.991,A -85,B 0,C 180,E1 -8903.56,E2 -8903.56} C_VEL
LIN {X 0,Y 438.364,Z 526.487,A -85,B 0,C 180,E1 -8905.402,E2 -8905.402} C_VEL
LIN {X 0,Y 438.379,Z 528.797,A -85,B 0,C 180,E1 -8907.243,E2 -8907.243} C_VEL
LIN {X 0,Y 438.252,Z 529.982,A -85,B 0,C 180,E1 -8909.081,E2 -8909.081} C_VEL
LIN {X 0,Y 438.253,Z 529.998,A -85,B 0,C 180,E1 -8910.919,E2 -8910.919} C_VEL
LIN {X 0,Y 438.379,Z 528.881,A -85,B 0,C 180,E1 -8912.757,E2 -8912.757} C_VEL
LIN {X 0,Y 438.361,Z 526.637,A -85,B 0,C 180,E1 -8914.598,E2 -8914.598} C_VEL
LIN {X 0,Y 438.545,Z 523.097,A -85,B 0,C 180,E1 -8916.488,E2 -8916.488} C_VEL
LIN {X 0,Y 438.812,Z 518.502,A -85,B 0,C 180,E1 -8918.287,E2 -8918.287} C_VEL
LIN {X 0,Y 439.163,Z 512.412,A -85,B 0,C 180,E1 -8920.139,E2 -8920.139} C_VEL
LIN {X 0,Y 439.799,Z 504.738,A -85,B 0,C 180,E1 -8921.99,E2 -8921.99} C_VEL
LIN {X 0,Y 440.407,Z 496.683,A -85,B 0,C 180,E1 -8923.59,E2 -8923.59} C_VEL
LIN {X 0,Y 441.283,Z 486.697,A -85,B 0,C 180,E1 -8925.235,E2 -8925.235} C_VEL
LIN {X 0,Y 442.146,Z 476.586,A -85,B 0,C 180,E1 -8926.625,E2 -8926.625} C_VEL
LIN {X 0,Y 443.139,Z 465.533,A -85,B 0,C 180,E1 -8927.903,E2 -8927.903} C_VEL
LIN {X 0,Y 444.193,Z 453.753,A -85,B 0,C 180,E1 -8929.046,E2 -8929.046} C_VEL
LIN {X 0,Y 445.216,Z 440.919,A -85,B 0,C 180,E1 -8930.08,E2 -8930.08} C_VEL
LIN {X 0,Y 446.226,Z 426.84,A -85,B 0,C 180,E1 -8930.996,E2 -8930.996} C_VEL
LIN {X 0,Y 447.038,Z 412.34,A -85,B 0,C 180,E1 -8931.736,E2 -8931.736} C_VEL
LIN {X 0,Y 447.67,Z 397.928,A -85,B 0,C 180,E1 -8932.285,E2 -8932.285} C_VEL
LIN {X 0,Y 448.111,Z 383.946,A -85,B 0,C 180,E1 -8932.657,E2 -8932.657} C_VEL
LIN {X 0,Y 449.68,Z 281.031,A -85,B 0,C 180,E1 -8934.35,E2 -8934.35} C_VEL
LIN {X 0,Y 450.072,Z 244.013,A -85,B 0,C 180,E1 -8934.965,E2 -8934.965} C_VEL
LIN {X 0,Y 447.102,Z 231.472,A -85,B 0,C 180,E1 -8935.362,E2 -8935.362} C_VEL
LIN {X 0,Y 442.493,Z 220.349,A -85,B 0,C 180,E1 -8935.863,E2 -8935.863} C_VEL
LIN {X 0,Y 439.954,Z 209.563,A -85,B 0,C 180,E1 -8938.069,E2 -8938.069} C_VEL
LIN {X 0,Y 439.425,Z 207.374,A -85,B 0,C 180,E1 -8938.537,E2 -8938.537} C_VEL
LIN {X 0,Y 439.369,Z 207.383,A -85,B 0,C 180,E1 -8942.03,E2 -8942.03} C_VEL
LIN {X 0,Y 439.393,Z 207.384,A -85,B 0,C 180,E1 -8945.34,E2 -8945.34} C_VEL
LIN {X 0,Y 439.386,Z 207.38,A -85,B 0,C 180,E1 -8948.594,E2 -8948.594} C_VEL
LIN {X 0,Y 439.386,Z 207.381,A -85,B 0,C 180,E1 -8951.256,E2 -8951.256} C_VEL
LIN {X 0,Y 439.401,Z 207.374,A -85,B 0,C 180,E1 -8954.728,E2 -8954.728} C_VEL
LIN {X 0,Y 439.392,Z 207.37,A -85,B 0,C 180,E1 -8957.795,E2 -8957.795} C_VEL
LIN {X 0,Y 439.445,Z 207.368,A -85,B 0,C 180,E1 -8960.229,E2 -8960.229} C_VEL
LIN {X 0,Y 439.371,Z 207.376,A -85,B 0,C 180,E1 -8963.712,E2 -8963.712} C_VEL
LIN {X 0,Y 439.366,Z 207.374,A -85,B 0,C 180,E1 -8967.053,E2 -8967.053} C_VEL
LIN {X 0,Y 439.389,Z 207.37,A -85,B 0,C 180,E1 -8970.275,E2 -8970.275} C_VEL
LIN {X 0,Y 439.421,Z 207.37,A -85,B 0,C 180,E1 -8973.396,E2 -8973.396} C_VEL
LIN {X 0,Y 439.379,Z 207.377,A -85,B 0,C 180,E1 -8976.429,E2 -8976.429} C_VEL
LIN {X 0,Y 439.381,Z 207.378,A -85,B 0,C 180,E1 -8979.397,E2 -8979.397} C_VEL
LIN {X 0,Y 439.423,Z 207.368,A -85,B 0,C 180,E1 -8982.309,E2 -8982.309} C_VEL
LIN {X 0,Y 439.439,Z 207.366,A -85,B 0,C 180,E1 -8985.174,E2 -8985.174} C_VEL
LIN {X 0,Y 439.476,Z 207.364,A -85,B 0,C 180,E1 -8988.001,E2 -8988.001} C_VEL
LIN {X 0,Y 439.539,Z 207.355,A -85,B 0,C 180,E1 -8991.726,E2 -8991.726} C_VEL
LIN {X 0,Y 439.612,Z 207.347,A -85,B 0,C 180,E1 -8994.496,E2 -8994.496} C_VEL
LIN {X 0,Y 439.627,Z 207.346,A -85,B 0,C 180,E1 -8998.168,E2 -8998.168} C_VEL
LIN {X 0,Y 439.755,Z 207.324,A -85,B 0,C 180,E1 -9000,E2 -9000} C_VEL
LIN {X 0,Y 439.647,Z 207.344,A -85,B 0,C 180,E1 -9002.749,E2 -9002.749} C_VEL
LIN {X 0,Y 439.609,Z 207.353,A -85,B 0,C 180,E1 -9006.425,E2 -9006.425} C_VEL
LIN {X 0,Y 439.492,Z 207.361,A -85,B 0,C 180,E1 -9009.202,E2 -9009.202} C_VEL
LIN {X 0,Y 439.457,Z 207.365,A -85,B 0,C 180,E1 -9012.938,E2 -9012.938} C_VEL
LIN {X 0,Y 439.452,Z 207.371,A -85,B 0,C 180,E1 -9016.355,E2 -9016.355} C_VEL
LIN {X 0,Y 439.394,Z 207.376,A -85,B 0,C 180,E1 -9019.627,E2 -9019.627} C_VEL
LIN {X 0,Y 439.357,Z 207.385,A -85,B 0,C 180,E1 -9022.576,E2 -9022.576} C_VEL
LIN {X 0,Y 439.397,Z 207.371,A -85,B 0,C 180,E1 -9025.585,E2 -9025.585} C_VEL
LIN {X 0,Y 439.418,Z 207.375,A -85,B 0,C 180,E1 -9028.673,E2 -9028.673} C_VEL
LIN {X 0,Y 439.375,Z 207.381,A -85,B 0,C 180,E1 -9032.034,E2 -9032.034} C_VEL
LIN {X 0,Y 439.389,Z 207.375,A -85,B 0,C 180,E1 -9035.341,E2 -9035.341} C_VEL
LIN {X 0,Y 439.372,Z 207.376,A -85,B 0,C 180,E1 -9038.596,E2 -9038.596} C_VEL
LIN {X 0,Y 439.382,Z 207.366,A -85,B 0,C 180,E1 -9041.257,E2 -9041.257} C_VEL
LIN {X 0,Y 439.396,Z 207.376,A -85,B 0,C 180,E1 -9044.73,E2 -9044.73} C_VEL
LIN {X 0,Y 439.392,Z 207.38,A -85,B 0,C 180,E1 -9047.796,E2 -9047.796} C_VEL
LIN {X 0,Y 439.445,Z 207.37,A -85,B 0,C 180,E1 -9050.23,E2 -9050.23} C_VEL
LIN {X 0,Y 439.373,Z 207.38,A -85,B 0,C 180,E1 -9053.714,E2 -9053.714} C_VEL
LIN {X 0,Y 439.369,Z 207.381,A -85,B 0,C 180,E1 -9057.055,E2 -9057.055} C_VEL
LIN {X 0,Y 439.406,Z 207.44,A -85,B 0,C 180,E1 -9058.177,E2 -9058.177} C_VEL
LIN {X 0,Y 443.214,Z 222.54,A -85,B 0,C 180,E1 -9060.992,E2 -9060.992} C_VEL
LIN {X 0,Y 444.951,Z 230.644,A -85,B 0,C 180,E1 -9062.435,E2 -9062.435} C_VEL
LIN {X 0,Y 444.145,Z 242.402,A -85,B 0,C 180,E1 -9064.294,E2 -9064.294} C_VEL
LIN {X 0,Y 449.929,Z 271.997,A -85,B 0,C 180,E1 -9065.156,E2 -9065.156} C_VEL
LIN {X 0,Y 447.857,Z 408.125,A -85,B 0,C 180,E1 -9067.39,E2 -9067.39} C_VEL
LIN {X 0,Y 447.287,Z 423.669,A -85,B 0,C 180,E1 -9067.816,E2 -9067.816} C_VEL
LIN {X 0,Y 446.471,Z 438.27,A -85,B 0,C 180,E1 -9068.394,E2 -9068.394} C_VEL
LIN {X 0,Y 445.612,Z 451.652,A -85,B 0,C 180,E1 -9069.095,E2 -9069.095} C_VEL
LIN {X 0,Y 444.569,Z 465.561,A -85,B 0,C 180,E1 -9070.01,E2 -9070.01} C_VEL
LIN {X 0,Y 443.537,Z 478.307,A -85,B 0,C 180,E1 -9071.045,E2 -9071.045} C_VEL
LIN {X 0,Y 442.529,Z 490.127,A -85,B 0,C 180,E1 -9072.199,E2 -9072.199} C_VEL
LIN {X 0,Y 441.491,Z 502,A -85,B 0,C 180,E1 -9073.587,E2 -9073.587} C_VEL
LIN {X 0,Y 440.606,Z 511.994,A -85,B 0,C 180,E1 -9074.978,E2 -9074.978} C_VEL
LIN {X 0,Y 439.761,Z 521.773,A -85,B 0,C 180,E1 -9076.601,E2 -9076.601} C_VEL
LIN {X 0,Y 439.234,Z 529.939,A -85,B 0,C 180,E1 -9078.229,E2 -9078.229} C_VEL
LIN {X 0,Y 438.774,Z 536.688,A -85,B 0,C 180,E1 -9079.852,E2 -9079.852} C_VEL
LIN {X 0,Y 438.54,Z 542.927,A -85,B 0,C 180,E1 -9081.707,E2 -9081.707} C_VEL
LIN {X 0,Y 438.363,Z 548.141,A -85,B 0,C 180,E1 -9083.723,E2 -9083.723} C_VEL
LIN {X 0,Y 438.283,Z 551.288,A -85,B 0,C 180,E1 -9085.401,E2 -9085.401} C_VEL
LIN {X 0,Y 438.324,Z 553.617,A -85,B 0,C 180,E1 -9087.243,E2 -9087.243} C_VEL
LIN {X 0,Y 438.249,Z 554.785,A -85,B 0,C 180,E1 -9089.081,E2 -9089.081} C_VEL
LIN {X 0,Y 438.249,Z 554.784,A -85,B 0,C 180,E1 -9090.919,E2 -9090.919} C_VEL
LIN {X 0,Y 438.324,Z 553.61,A -85,B 0,C 180,E1 -9092.757,E2 -9092.757} C_VEL
LIN {X 0,Y 438.285,Z 551.28,A -85,B 0,C 180,E1 -9094.599,E2 -9094.599} C_VEL
LIN {X 0,Y 438.395,Z 547.749,A -85,B 0,C 180,E1 -9096.443,E2 -9096.443} C_VEL
LIN {X 0,Y 438.54,Z 542.923,A -85,B 0,C 180,E1 -9098.293,E2 -9098.293} C_VEL
LIN {X 0,Y 438.774,Z 536.674,A -85,B 0,C 180,E1 -9100.148,E2 -9100.148} C_VEL
LIN {X 0,Y 439.232,Z 529.92,A -85,B 0,C 180,E1 -9101.771,E2 -9101.771} C_VEL
LIN {X 0,Y 439.758,Z 521.755,A -85,B 0,C 180,E1 -9103.399,E2 -9103.399} C_VEL
LIN {X 0,Y 440.611,Z 511.973,A -85,B 0,C 180,E1 -9105.022,E2 -9105.022} C_VEL
LIN {X 0,Y 441.508,Z 501.974,A -85,B 0,C 180,E1 -9106.412,E2 -9106.412} C_VEL
LIN {X 0,Y 442.369,Z 492.031,A -85,B 0,C 180,E1 -9107.593,E2 -9107.593} C_VEL
LIN {X 0,Y 443.404,Z 479.568,A -85,B 0,C 180,E1 -9108.841,E2 -9108.841} C_VEL
LIN {X 0,Y 444.445,Z 467.089,A -85,B 0,C 180,E1 -9109.875,E2 -9109.875} C_VEL
LIN {X 0,Y 445.467,Z 453.565,A -85,B 0,C 180,E1 -9110.791,E2 -9110.791} C_VEL
LIN {X 0,Y 446.463,Z 439.069,A -85,B 0,C 180,E1 -9111.565,E2 -9111.565} C_VEL
LIN {X 0,Y 447.209,Z 423.549,A -85,B 0,C 180,E1 -9112.188,E2 -9112.188} C_VEL
LIN {X 0,Y 447.86,Z 407.899,A -85,B 0,C 180,E1 -9112.61,E2 -9112.61} C_VEL
LIN {X 0,Y 449.942,Z 272.064,A -85,B 0,C 180,E1 -9114.837,E2 -9114.837} C_VEL
LIN {X 0,Y 444.185,Z 242.352,A -85,B 0,C 180,E1 -9115.705,E2 -9115.705} C_VEL
LIN {X 0,Y 444.942,Z 230.619,A -85,B 0,C 180,E1 -9117.563,E2 -9117.563} C_VEL
LIN {X 0,Y 442.569,Z 219.853,A -85,B 0,C 180,E1 -9119.49,E2 -9119.49} C_VEL
LIN {X 0,Y 439.37,Z 207.374,A -85,B 0,C 180,E1 -9121.86,E2 -9121.86} C_VEL
LIN {X 0,Y 439.397,Z 207.371,A -85,B 0,C 180,E1 -9125.155,E2 -9125.155} C_VEL
LIN {X 0,Y 439.392,Z 207.378,A -85,B 0,C 180,E1 -9128.593,E2 -9128.593} C_VEL
LIN {X 0,Y 439.394,Z 207.375,A -85,B 0,C 180,E1 -9131.258,E2 -9131.258} C_VEL
LIN {X 0,Y 439.396,Z 207.372,A -85,B 0,C 180,E1 -9134.729,E2 -9134.729} C_VEL
LIN {X 0,Y 439.392,Z 207.376,A -85,B 0,C 180,E1 -9137.795,E2 -9137.795} C_VEL
LIN {X 0,Y 439.443,Z 207.369,A -85,B 0,C 180,E1 -9140.229,E2 -9140.229} C_VEL
LIN {X 0,Y 439.37,Z 207.379,A -85,B 0,C 180,E1 -9143.713,E2 -9143.713} C_VEL
LIN {X 0,Y 439.368,Z 207.373,A -85,B 0,C 180,E1 -9147.054,E2 -9147.054} C_VEL
LIN {X 0,Y 439.389,Z 207.374,A -85,B 0,C 180,E1 -9150.275,E2 -9150.275} C_VEL
LIN {X 0,Y 439.426,Z 207.371,A -85,B 0,C 180,E1 -9153.588,E2 -9153.588} C_VEL
LIN {X 0,Y 439.378,Z 207.372,A -85,B 0,C 180,E1 -9156.429,E2 -9156.429} C_VEL
LIN {X 0,Y 439.38,Z 207.366,A -85,B 0,C 180,E1 -9159.397,E2 -9159.397} C_VEL
LIN {X 0,Y 439.423,Z 207.37,A -85,B 0,C 180,E1 -9162.309,E2 -9162.309} C_VEL
LIN {X 0,Y 439.439,Z 207.37,A -85,B 0,C 180,E1 -9165.174,E2 -9165.174} C_VEL
LIN {X 0,Y 439.475,Z 207.365,A -85,B 0,C 180,E1 -9168.001,E2 -9168.001} C_VEL
LIN {X 0,Y 439.539,Z 207.357,A -85,B 0,C 180,E1 -9171.726,E2 -9171.726} C_VEL
LIN {X 0,Y 439.613,Z 207.346,A -85,B 0,C 180,E1 -9174.496,E2 -9174.496} C_VEL
LIN {X 0,Y 439.627,Z 207.345,A -85,B 0,C 180,E1 -9178.168,E2 -9178.168} C_VEL
LIN {X 0,Y 439.755,Z 207.326,A -85,B 0,C 180,E1 -9180,E2 -9180} C_VEL
LIN {X 0,Y 439.648,Z 207.344,A -85,B 0,C 180,E1 -9182.749,E2 -9182.749} C_VEL
LIN {X 0,Y 439.611,Z 207.347,A -85,B 0,C 180,E1 -9186.425,E2 -9186.425} C_VEL
LIN {X 0,Y 439.492,Z 207.363,A -85,B 0,C 180,E1 -9189.202,E2 -9189.202} C_VEL
LIN {X 0,Y 439.461,Z 207.366,A -85,B 0,C 180,E1 -9192.938,E2 -9192.938} C_VEL
LIN {X 0,Y 439.439,Z 207.367,A -85,B 0,C 180,E1 -9196.349,E2 -9196.349} C_VEL
LIN {X 0,Y 439.394,Z 207.374,A -85,B 0,C 180,E1 -9199.627,E2 -9199.627} C_VEL
LIN {X 0,Y 439.357,Z 207.38,A -85,B 0,C 180,E1 -9202.576,E2 -9202.576} C_VEL
LIN {X 0,Y 439.397,Z 207.358,A -85,B 0,C 180,E1 -9205.585,E2 -9205.585} C_VEL
LIN {X 0,Y 439.419,Z 207.372,A -85,B 0,C 180,E1 -9208.673,E2 -9208.673} C_VEL
LIN {X 0,Y 439.368,Z 207.377,A -85,B 0,C 180,E1 -9211.861,E2 -9211.861} C_VEL
LIN {X 0,Y 439.395,Z 207.377,A -85,B 0,C 180,E1 -9215.157,E2 -9215.157} C_VEL
LIN {X 0,Y 439.378,Z 207.379,A -85,B 0,C 180,E1 -9218.596,E2 -9218.596} C_VEL
LIN {X 0,Y 439.384,Z 207.374,A -85,B 0,C 180,E1 -9221.257,E2 -9221.257} C_VEL
LIN {X 0,Y 439.402,Z 207.376,A -85,B 0,C 180,E1 -9224.729,E2 -9224.729} C_VEL
LIN {X 0,Y 439.394,Z 207.375,A -85,B 0,C 180,E1 -9227.797,E2 -9227.797} C_VEL
LIN {X 0,Y 439.434,Z 207.373,A -85,B 0,C 180,E1 -9230.229,E2 -9230.229} C_VEL
LIN {X 0,Y 439.371,Z 207.377,A -85,B 0,C 180,E1 -9233.714,E2 -9233.714} C_VEL
LIN {X 0,Y 439.371,Z 207.379,A -85,B 0,C 180,E1 -9237.055,E2 -9237.055} C_VEL
LIN {X 0,Y 439.381,Z 207.38,A -85,B 0,C 180,E1 -9240.275,E2 -9240.275} C_VEL
LIN {X 0,Y 439.447,Z 207.503,A -85,B 0,C 180,E1 -9241.595,E2 -9241.595} C_VEL
LIN {X 0,Y 442.257,Z 219.318,A -85,B 0,C 180,E1 -9244.025,E2 -9244.025} C_VEL
LIN {X 0,Y 442.584,Z 220.762,A -85,B 0,C 180,E1 -9244.265,E2 -9244.265} C_VEL
LIN {X 0,Y 447.656,Z 233.422,A -85,B 0,C 180,E1 -9244.801,E2 -9244.801} C_VEL
LIN {X 0,Y 450.08,Z 244.11,A -85,B 0,C 180,E1 -9245.132,E2 -9245.132} C_VEL
LIN {X 0,Y 448.619,Z 352.72,A -85,B 0,C 180,E1 -9246.913,E2 -9246.913} C_VEL
LIN {X 0,Y 448.048,Z 386.448,A -85,B 0,C 180,E1 -9247.491,E2 -9247.491} C_VEL
LIN {X 0,Y 447.559,Z 401.745,A -85,B 0,C 180,E1 -9247.936,E2 -9247.936} C_VEL
LIN {X 0,Y 447.091,Z 405.587,A -85,B 0,C 180,E1 -9248.064,E2 -9248.064} C_VEL
LIN {X 0,Y 444.943,Z 413.148,A -85,B 0,C 180,E1 -9248.283,E2 -9248.283} C_VEL
LIN {X 0,Y 440.307,Z 425.72,A -85,B 0,C 180,E1 -9248.721,E2 -9248.721} C_VEL
LIN {X 0,Y 439.282,Z 430.99,A -85,B 0,C 180,E1 -9249.002,E2 -9249.002} C_VEL
LIN {X 0,Y 438.274,Z 444.596,A -85,B 0,C 180,E1 -9249.955,E2 -9249.955} C_VEL
LIN {X 0,Y 437.076,Z 458.066,A -85,B 0,C 180,E1 -9251.12,E2 -9251.12} C_VEL
LIN {X 0,Y 436.01,Z 470.278,A -85,B 0,C 180,E1 -9252.409,E2 -9252.409} C_VEL
LIN {X 0,Y 434.921,Z 481.4,A -85,B 0,C 180,E1 -9253.815,E2 -9253.815} C_VEL
LIN {X 0,Y 433.892,Z 492.201,A -85,B 0,C 180,E1 -9255.46,E2 -9255.46} C_VEL
LIN {X 0,Y 433.036,Z 500.716,A -85,B 0,C 180,E1 -9257.018,E2 -9257.018} C_VEL
LIN {X 0,Y 432.59,Z 507.584,A -85,B 0,C 180,E1 -9258.521,E2 -9258.521} C_VEL
LIN {X 0,Y 432.045,Z 513.925,A -85,B 0,C 180,E1 -9260.166,E2 -9260.166} C_VEL
LIN {X 0,Y 431.684,Z 519.747,A -85,B 0,C 180,E1 -9262.046,E2 -9262.046} C_VEL
LIN {X 0,Y 431.522,Z 523.193,A -85,B 0,C 180,E1 -9263.454,E2 -9263.454} C_VEL
LIN {X 0,Y 431.294,Z 526.689,A -85,B 0,C 180,E1 -9265.327,E2 -9265.327} C_VEL
LIN {X 0,Y 431.307,Z 528.997,A -85,B 0,C 180,E1 -9267.198,E2 -9267.198} C_VEL
LIN {X 0,Y 431.169,Z 530.182,A -85,B 0,C 180,E1 -9269.066,E2 -9269.066} C_VEL
LIN {X 0,Y 431.17,Z 530.199,A -85,B 0,C 180,E1 -9270.934,E2 -9270.934} C_VEL
LIN {X 0,Y 431.307,Z 529.081,A -85,B 0,C 180,E1 -9272.802,E2 -9272.802} C_VEL
LIN {X 0,Y 431.29,Z 526.837,A -85,B 0,C 180,E1 -9274.673,E2 -9274.673} C_VEL
LIN {X 0,Y 431.481,Z 523.403,A -85,B 0,C 180,E1 -9276.547,E2 -9276.547} C_VEL
LIN {X 0,Y 431.755,Z 518.703,A -85,B 0,C 180,E1 -9278.424,E2 -9278.424} C_VEL
LIN {X 0,Y 432.128,Z 512.612,A -85,B 0,C 180,E1 -9280.305,E2 -9280.305} C_VEL
LIN {X 0,Y 432.826,Z 504.937,A -85,B 0,C 180,E1 -9282.186,E2 -9282.186} C_VEL
LIN {X 0,Y 433.444,Z 496.883,A -85,B 0,C 180,E1 -9283.813,E2 -9283.813} C_VEL
LIN {X 0,Y 434.386,Z 486.897,A -85,B 0,C 180,E1 -9285.483,E2 -9285.483} C_VEL
LIN {X 0,Y 435.309,Z 476.785,A -85,B 0,C 180,E1 -9286.894,E2 -9286.894} C_VEL
LIN {X 0,Y 436.47,Z 464.773,A -85,B 0,C 180,E1 -9288.296,E2 -9288.296} C_VEL
LIN {X 0,Y 437.594,Z 452.664,A -85,B 0,C 180,E1 -9289.466,E2 -9289.466} C_VEL
LIN {X 0,Y 438.647,Z 439.54,A -85,B 0,C 180,E1 -9290.516,E2 -9290.516} C_VEL
LIN {X 0,Y 439.599,Z 427.034,A -85,B 0,C 180,E1 -9291.328,E2 -9291.328} C_VEL
LIN {X 0,Y 440.441,Z 412.866,A -85,B 0,C 180,E1 -9292.062,E2 -9292.062} C_VEL
LIN {X 0,Y 441.124,Z 398.115,A -85,B 0,C 180,E1 -9292.634,E2 -9292.634} C_VEL
LIN {X 0,Y 441.59,Z 384.124,A -85,B 0,C 180,E1 -9293.011,E2 -9293.011} C_VEL
LIN {X 0,Y 443.235,Z 282.243,A -85,B 0,C 180,E1 -9294.71,E2 -9294.71} C_VEL
LIN {X 0,Y 443.654,Z 245.264,A -85,B 0,C 180,E1 -9295.333,E2 -9295.333} C_VEL
LIN {X 0,Y 440.902,Z 233.861,A -85,B 0,C 180,E1 -9295.705,E2 -9295.705} C_VEL
LIN {X 0,Y 435.334,Z 220.585,A -85,B 0,C 180,E1 -9296.317,E2 -9296.317} C_VEL
LIN {X 0,Y 432.377,Z 208.252,A -85,B 0,C 180,E1 -9298.922,E2 -9298.922} C_VEL
LIN {X 0,Y 432.321,Z 208.259,A -85,B 0,C 180,E1 -9302.442,E2 -9302.442} C_VEL
LIN {X 0,Y 432.343,Z 208.259,A -85,B 0,C 180,E1 -9305.631,E2 -9305.631} C_VEL
LIN {X 0,Y 432.348,Z 208.257,A -85,B 0,C 180,E1 -9308.715,E2 -9308.715} C_VEL
LIN {X 0,Y 432.332,Z 208.257,A -85,B 0,C 180,E1 -9311.796,E2 -9311.796} C_VEL
LIN {X 0,Y 432.336,Z 208.253,A -85,B 0,C 180,E1 -9314.346,E2 -9314.346} C_VEL
LIN {X 0,Y 432.316,Z 208.253,A -85,B 0,C 180,E1 -9317.015,E2 -9317.015} C_VEL
LIN {X 0,Y 432.351,Z 208.253,A -85,B 0,C 180,E1 -9319.817,E2 -9319.817} C_VEL
LIN {X 0,Y 432.311,Z 208.248,A -85,B 0,C 180,E1 -9323.022,E2 -9323.022} C_VEL
LIN {X 0,Y 432.353,Z 208.251,A -85,B 0,C 180,E1 -9325.996,E2 -9325.996} C_VEL
LIN {X 0,Y 432.388,Z 208.243,A -85,B 0,C 180,E1 -9329.743,E2 -9329.743} C_VEL
LIN {X 0,Y 432.392,Z 208.246,A -85,B 0,C 180,E1 -9333.372,E2 -9333.372} C_VEL
LIN {X 0,Y 432.364,Z 208.25,A -85,B 0,C 180,E1 -9336.023,E2 -9336.023} C_VEL
LIN {X 0,Y 432.342,Z 208.259,A -85,B 0,C 180,E1 -9339.046,E2 -9339.046} C_VEL
LIN {X 0,Y 432.37,Z 208.245,A -85,B 0,C 180,E1 -9342.011,E2 -9342.011} C_VEL
LIN {X 0,Y 432.387,Z 208.247,A -85,B 0,C 180,E1 -9344.926,E2 -9344.926} C_VEL
LIN {X 0,Y 432.451,Z 208.239,A -85,B 0,C 180,E1 -9347.803,E2 -9347.803} C_VEL
LIN {X 0,Y 432.483,Z 208.235,A -85,B 0,C 180,E1 -9351.59,E2 -9351.59} C_VEL
LIN {X 0,Y 432.589,Z 208.223,A -85,B 0,C 180,E1 -9354.406,E2 -9354.406} C_VEL
LIN {X 0,Y 432.597,Z 208.222,A -85,B 0,C 180,E1 -9358.138,E2 -9358.138} C_VEL
LIN {X 0,Y 432.725,Z 208.2,A -85,B 0,C 180,E1 -9360,E2 -9360} C_VEL
LIN {X 0,Y 432.597,Z 208.222,A -85,B 0,C 180,E1 -9362.793,E2 -9362.793} C_VEL
LIN {X 0,Y 432.564,Z 208.232,A -85,B 0,C 180,E1 -9366.53,E2 -9366.53} C_VEL
LIN {X 0,Y 432.435,Z 208.24,A -85,B 0,C 180,E1 -9369.353,E2 -9369.353} C_VEL
LIN {X 0,Y 432.422,Z 208.242,A -85,B 0,C 180,E1 -9372.804,E2 -9372.804} C_VEL
LIN {X 0,Y 432.414,Z 208.246,A -85,B 0,C 180,E1 -9376.484,E2 -9376.484} C_VEL
LIN {X 0,Y 432.331,Z 208.259,A -85,B 0,C 180,E1 -9379.961,E2 -9379.961} C_VEL
LIN {X 0,Y 432.311,Z 208.259,A -85,B 0,C 180,E1 -9382.965,E2 -9382.965} C_VEL
LIN {X 0,Y 432.356,Z 208.251,A -85,B 0,C 180,E1 -9386.033,E2 -9386.033} C_VEL
LIN {X 0,Y 432.345,Z 208.253,A -85,B 0,C 180,E1 -9389.187,E2 -9389.187} C_VEL
LIN {X 0,Y 432.324,Z 208.256,A -85,B 0,C 180,E1 -9392.295,E2 -9392.295} C_VEL
LIN {X 0,Y 432.334,Z 208.255,A -85,B 0,C 180,E1 -9394.677,E2 -9394.677} C_VEL
LIN {X 0,Y 432.331,Z 208.258,A -85,B 0,C 180,E1 -9398.15,E2 -9398.15} C_VEL
LIN {X 0,Y 432.326,Z 208.247,A -85,B 0,C 180,E1 -9401.603,E2 -9401.603} C_VEL
LIN {X 0,Y 432.328,Z 208.257,A -85,B 0,C 180,E1 -9404.348,E2 -9404.348} C_VEL
LIN {X 0,Y 432.315,Z 208.257,A -85,B 0,C 180,E1 -9407.016,E2 -9407.016} C_VEL
LIN {X 0,Y 432.351,Z 208.255,A -85,B 0,C 180,E1 -9409.818,E2 -9409.818} C_VEL
LIN {X 0,Y 432.312,Z 208.254,A -85,B 0,C 180,E1 -9413.024,E2 -9413.024} C_VEL
LIN {X 0,Y 432.356,Z 208.256,A -85,B 0,C 180,E1 -9415.997,E2 -9415.997} C_VEL
LIN {X 0,Y 432.324,Z 208.296,A -85,B 0,C 180,E1 -9417.778,E2 -9417.778} C_VEL
LIN {X 0,Y 435.789,Z 221.747,A -85,B 0,C 180,E1 -9420.352,E2 -9420.352} C_VEL
LIN {X 0,Y 438.135,Z 232.308,A -85,B 0,C 180,E1 -9422.279,E2 -9422.279} C_VEL
LIN {X 0,Y 437.492,Z 242.446,A -85,B 0,C 180,E1 -9423.878,E2 -9423.878} C_VEL
LIN {X 0,Y 443.467,Z 272.978,A -85,B 0,C 180,E1 -9424.789,E2 -9424.789} C_VEL
LIN {X 0,Y 441.308,Z 407.939,A -85,B 0,C 180,E1 -9427.035,E2 -9427.035} C_VEL
LIN {X 0,Y 440.696,Z 423.477,A -85,B 0,C 180,E1 -9427.466,E2 -9427.466} C_VEL
LIN {X 0,Y 439.871,Z 438.167,A -85,B 0,C 180,E1 -9428.058,E2 -9428.058} C_VEL
LIN {X 0,Y 438.973,Z 451.456,A -85,B 0,C 180,E1 -9428.763,E2 -9428.763} C_VEL
LIN {X 0,Y 437.845,Z 465.362,A -85,B 0,C 180,E1 -9429.69,E2 -9429.69} C_VEL
LIN {X 0,Y 436.798,Z 478.109,A -85,B 0,C 180,E1 -9430.741,E2 -9430.741} C_VEL
LIN {X 0,Y 435.692,Z 489.926,A -85,B 0,C 180,E1 -9431.91,E2 -9431.91} C_VEL
LIN {X 0,Y 434.633,Z 501.8,A -85,B 0,C 180,E1 -9433.321,E2 -9433.321} C_VEL
LIN {X 0,Y 433.671,Z 511.792,A -85,B 0,C 180,E1 -9434.732,E2 -9434.732} C_VEL
LIN {X 0,Y 432.794,Z 521.572,A -85,B 0,C 180,E1 -9436.382,E2 -9436.382} C_VEL
LIN {X 0,Y 432.216,Z 529.737,A -85,B 0,C 180,E1 -9438.035,E2 -9438.035} C_VEL
LIN {X 0,Y 431.731,Z 536.487,A -85,B 0,C 180,E1 -9439.685,E2 -9439.685} C_VEL
LIN {X 0,Y 431.45,Z 542.725,A -85,B 0,C 180,E1 -9441.57,E2 -9441.57} C_VEL
LIN {X 0,Y 431.287,Z 547.552,A -85,B 0,C 180,E1 -9443.45,E2 -9443.45} C_VEL
LIN {X 0,Y 431.208,Z 551.088,A -85,B 0,C 180,E1 -9445.326,E2 -9445.326} C_VEL
LIN {X 0,Y 431.217,Z 553.416,A -85,B 0,C 180,E1 -9447.198,E2 -9447.198} C_VEL
LIN {X 0,Y 431.166,Z 554.585,A -85,B 0,C 180,E1 -9449.066,E2 -9449.066} C_VEL
LIN {X 0,Y 431.166,Z 554.584,A -85,B 0,C 180,E1 -9450.934,E2 -9450.934} C_VEL
LIN {X 0,Y 431.217,Z 553.409,A -85,B 0,C 180,E1 -9452.802,E2 -9452.802} C_VEL
LIN {X 0,Y 431.21,Z 551.079,A -85,B 0,C 180,E1 -9454.674,E2 -9454.674} C_VEL
LIN {X 0,Y 431.324,Z 547.547,A -85,B 0,C 180,E1 -9456.549,E2 -9456.549} C_VEL
LIN {X 0,Y 431.45,Z 542.72,A -85,B 0,C 180,E1 -9458.43,E2 -9458.43} C_VEL
LIN {X 0,Y 431.73,Z 536.47,A -85,B 0,C 180,E1 -9460.315,E2 -9460.315} C_VEL
LIN {X 0,Y 432.203,Z 529.715,A -85,B 0,C 180,E1 -9461.965,E2 -9461.965} C_VEL
LIN {X 0,Y 432.899,Z 520.287,A -85,B 0,C 180,E1 -9463.854,E2 -9463.854} C_VEL
LIN {X 0,Y 433.809,Z 510.245,A -85,B 0,C 180,E1 -9465.504,E2 -9465.504} C_VEL
LIN {X 0,Y 434.806,Z 499.977,A -85,B 0,C 180,E1 -9466.914,E2 -9466.914} C_VEL
LIN {X 0,Y 435.889,Z 487.745,A -85,B 0,C 180,E1 -9468.324,E2 -9468.324} C_VEL
LIN {X 0,Y 437.017,Z 475.473,A -85,B 0,C 180,E1 -9469.493,E2 -9469.493} C_VEL
LIN {X 0,Y 438.12,Z 462.12,A -85,B 0,C 180,E1 -9470.542,E2 -9470.542} C_VEL
LIN {X 0,Y 439.252,Z 447.387,A -85,B 0,C 180,E1 -9471.469,E2 -9471.469} C_VEL
LIN {X 0,Y 440.183,Z 432.8,A -85,B 0,C 180,E1 -9472.176,E2 -9472.176} C_VEL
LIN {X 0,Y 440.895,Z 418.753,A -85,B 0,C 180,E1 -9472.678,E2 -9472.678} C_VEL
LIN {X 0,Y 441.414,Z 403.161,A -85,B 0,C 180,E1 -9473.052,E2 -9473.052} C_VEL
LIN {X 0,Y 443.425,Z 272.452,A -85,B 0,C 180,E1 -9475.217,E2 -9475.217} C_VEL
LIN {X 0,Y 437.463,Z 242.004,A -85,B 0,C 180,E1 -9476.152,E2 -9476.152} C_VEL
LIN {X 0,Y 438.136,Z 232.266,A -85,B 0,C 180,E1 -9477.721,E2 -9477.721} C_VEL
LIN {X 0,Y 435.515,Z 220.665,A -85,B 0,C 180,E1 -9479.842,E2 -9479.842} C_VEL
LIN {X 0,Y 432.324,Z 208.254,A -85,B 0,C 180,E1 -9482.222,E2 -9482.222} C_VEL
LIN {X 0,Y 432.337,Z 208.252,A -85,B 0,C 180,E1 -9484.676,E2 -9484.676} C_VEL
LIN {X 0,Y 432.347,Z 208.258,A -85,B 0,C 180,E1 -9488.148,E2 -9488.148} C_VEL
LIN {X 0,Y 432.362,Z 208.252,A -85,B 0,C 180,E1 -9491.606,E2 -9491.606} C_VEL
LIN {X 0,Y 432.329,Z 208.256,A -85,B 0,C 180,E1 -9494.347,E2 -9494.347} C_VEL
LIN {X 0,Y 432.315,Z 208.254,A -85,B 0,C 180,E1 -9497.015,E2 -9497.015} C_VEL
LIN {X 0,Y 432.349,Z 208.252,A -85,B 0,C 180,E1 -9499.817,E2 -9499.817} C_VEL
LIN {X 0,Y 432.31,Z 208.254,A -85,B 0,C 180,E1 -9503.022,E2 -9503.022} C_VEL
LIN {X 0,Y 432.353,Z 208.252,A -85,B 0,C 180,E1 -9505.996,E2 -9505.996} C_VEL
LIN {X 0,Y 432.388,Z 208.248,A -85,B 0,C 180,E1 -9509.744,E2 -9509.744} C_VEL
LIN {X 0,Y 432.392,Z 208.246,A -85,B 0,C 180,E1 -9513.372,E2 -9513.372} C_VEL
LIN {X 0,Y 432.363,Z 208.249,A -85,B 0,C 180,E1 -9516.023,E2 -9516.023} C_VEL
LIN {X 0,Y 432.342,Z 208.239,A -85,B 0,C 180,E1 -9519.046,E2 -9519.046} C_VEL
LIN {X 0,Y 432.37,Z 208.251,A -85,B 0,C 180,E1 -9522.011,E2 -9522.011} C_VEL
LIN {X 0,Y 432.386,Z 208.247,A -85,B 0,C 180,E1 -9524.926,E2 -9524.926} C_VEL
LIN {X 0,Y 432.451,Z 208.24,A -85,B 0,C 180,E1 -9527.803,E2 -9527.803} C_VEL
LIN {X 0,Y 432.483,Z 208.236,A -85,B 0,C 180,E1 -9531.59,E2 -9531.59} C_VEL
LIN {X 0,Y 432.589,Z 208.221,A -85,B 0,C 180,E1 -9534.406,E2 -9534.406} C_VEL
LIN {X 0,Y 432.597,Z 208.221,A -85,B 0,C 180,E1 -9538.138,E2 -9538.138} C_VEL
LIN {X 0,Y 432.726,Z 208.201,A -85,B 0,C 180,E1 -9540,E2 -9540} C_VEL
LIN {X 0,Y 432.597,Z 208.222,A -85,B 0,C 180,E1 -9542.794,E2 -9542.794} C_VEL
LIN {X 0,Y 432.565,Z 208.225,A -85,B 0,C 180,E1 -9546.531,E2 -9546.531} C_VEL
LIN {X 0,Y 432.435,Z 208.243,A -85,B 0,C 180,E1 -9549.353,E2 -9549.353} C_VEL
LIN {X 0,Y 432.424,Z 208.242,A -85,B 0,C 180,E1 -9552.805,E2 -9552.805} C_VEL
LIN {X 0,Y 432.404,Z 208.243,A -85,B 0,C 180,E1 -9556.479,E2 -9556.479} C_VEL
LIN {X 0,Y 432.33,Z 208.252,A -85,B 0,C 180,E1 -9559.961,E2 -9559.961} C_VEL
LIN {X 0,Y 432.311,Z 208.262,A -85,B 0,C 180,E1 -9562.965,E2 -9562.965} C_VEL
LIN {X 0,Y 432.357,Z 208.232,A -85,B 0,C 180,E1 -9566.033,E2 -9566.033} C_VEL
LIN {X 0,Y 432.346,Z 208.257,A -85,B 0,C 180,E1 -9569.187,E2 -9569.187} C_VEL
LIN {X 0,Y 432.319,Z 208.256,A -85,B 0,C 180,E1 -9572.294,E2 -9572.294} C_VEL
LIN {X 0,Y 432.335,Z 208.254,A -85,B 0,C 180,E1 -9574.678,E2 -9574.678} C_VEL
LIN {X 0,Y 432.34,Z 208.252,A -85,B 0,C 180,E1 -9578.15,E2 -9578.15} C_VEL
LIN {X 0,Y 432.328,Z 208.251,A -85,B 0,C 180,E1 -9581.603,E2 -9581.603} C_VEL
LIN {X 0,Y 432.337,Z 208.254,A -85,B 0,C 180,E1 -9584.347,E2 -9584.347} C_VEL
LIN {X 0,Y 432.321,Z 208.261,A -85,B 0,C 180,E1 -9587.016,E2 -9587.016} C_VEL
LIN {X 0,Y 432.338,Z 208.255,A -85,B 0,C 180,E1 -9589.82,E2 -9589.82} C_VEL
LIN {X 0,Y 432.304,Z 208.261,A -85,B 0,C 180,E1 -9593.023,E2 -9593.023} C_VEL
LIN {X 0,Y 432.357,Z 208.255,A -85,B 0,C 180,E1 -9595.997,E2 -9595.997} C_VEL
LIN {X 0,Y 432.346,Z 208.257,A -85,B 0,C 180,E1 -9599.49,E2 -9599.49} C_VEL
LIN {X 0,Y 432.393,Z 208.376,A -85,B 0,C 180,E1 -9601.22,E2 -9601.22} C_VEL
LIN {X 0,Y 435.208,Z 220.042,A -85,B 0,C 180,E1 -9603.668,E2 -9603.668} C_VEL
LIN {X 0,Y 435.431,Z 220.994,A -85,B 0,C 180,E1 -9603.81,E2 -9603.81} C_VEL
LIN {X 0,Y 441.533,Z 235.941,A -85,B 0,C 180,E1 -9604.468,E2 -9604.468} C_VEL
LIN {X 0,Y 443.717,Z 246.04,A -85,B 0,C 180,E1 -9604.781,E2 -9604.781} C_VEL
LIN {X 0,Y 442.115,Z 352.947,A -85,B 0,C 180,E1 -9606.553,E2 -9606.553} C_VEL
LIN {X 0,Y 441.515,Z 386.665,A -85,B 0,C 180,E1 -9607.14,E2 -9607.14} C_VEL
LIN {X 0,Y 440.98,Z 402.215,A -85,B 0,C 180,E1 -9607.599,E2 -9607.599} C_VEL
LIN {X 0,Y 440.277,Z 416.373,A -85,B 0,C 180,E1 -9608.193,E2 -9608.193} C_VEL
LIN {X 0,Y 439.282,Z 430.99,A -85,B 0,C 180,E1 -9609.002,E2 -9609.002} C_VEL
LIN {X 0,Y 438.253,Z 436.316,A -85,B 0,C 180,E1 -9609.314,E2 -9609.314} C_VEL
LIN {X 0,Y 434.873,Z 444.88,A -85,B 0,C 180,E1 -9609.807,E2 -9609.807} C_VEL
LIN {X 0,Y 431.46,Z 453.172,A -85,B 0,C 180,E1 -9610.369,E2 -9610.369} C_VEL
LIN {X 0,Y 430.379,Z 457.989,A -85,B 0,C 180,E1 -9610.786,E2 -9610.786} C_VEL
LIN {X 0,Y 429.235,Z 470.483,A -85,B 0,C 180,E1 -9612.122,E2 -9612.122} C_VEL
LIN {X 0,Y 428.069,Z 481.606,A -85,B 0,C 180,E1 -9613.549,E2 -9613.549} C_VEL
LIN {X 0,Y 426.993,Z 492.406,A -85,B 0,C 180,E1 -9615.22,E2 -9615.22} C_VEL
LIN {X 0,Y 426.054,Z 501.33,A -85,B 0,C 180,E1 -9616.883,E2 -9616.883} C_VEL
LIN {X 0,Y 425.495,Z 508.788,A -85,B 0,C 180,E1 -9618.568,E2 -9618.568} C_VEL
LIN {X 0,Y 424.916,Z 515.728,A -85,B 0,C 180,E1 -9620.48,E2 -9620.48} C_VEL
LIN {X 0,Y 424.547,Z 521.18,A -85,B 0,C 180,E1 -9622.39,E2 -9622.39} C_VEL
LIN {X 0,Y 424.352,Z 525.295,A -85,B 0,C 180,E1 -9624.297,E2 -9624.297} C_VEL
LIN {X 0,Y 424.155,Z 528.19,A -85,B 0,C 180,E1 -9626.2,E2 -9626.2} C_VEL
LIN {X 0,Y 424.149,Z 529.93,A -85,B 0,C 180,E1 -9628.101,E2 -9628.101} C_VEL
LIN {X 0,Y 424.083,Z 530.54,A -85,B 0,C 180,E1 -9630,E2 -9630} C_VEL
LIN {X 0,Y 424.149,Z 529.979,A -85,B 0,C 180,E1 -9631.899,E2 -9631.899} C_VEL
LIN {X 0,Y 424.154,Z 528.305,A -85,B 0,C 180,E1 -9633.8,E2 -9633.8} C_VEL
LIN {X 0,Y 424.336,Z 525.472,A -85,B 0,C 180,E1 -9635.703,E2 -9635.703} C_VEL
LIN {X 0,Y 424.541,Z 521.418,A -85,B 0,C 180,E1 -9637.61,E2 -9637.61} C_VEL
LIN {X 0,Y 424.904,Z 516.041,A -85,B 0,C 180,E1 -9639.52,E2 -9639.52} C_VEL
LIN {X 0,Y 425.481,Z 509.187,A -85,B 0,C 180,E1 -9641.432,E2 -9641.432} C_VEL
LIN {X 0,Y 426.036,Z 501.831,A -85,B 0,C 180,E1 -9643.107,E2 -9643.107} C_VEL
LIN {X 0,Y 426.936,Z 492.93,A -85,B 0,C 180,E1 -9644.782,E2 -9644.782} C_VEL
LIN {X 0,Y 427.871,Z 483.868,A -85,B 0,C 180,E1 -9646.214,E2 -9646.214} C_VEL
LIN {X 0,Y 428.714,Z 475.119,A -85,B 0,C 180,E1 -9647.408,E2 -9647.408} C_VEL
LIN {X 0,Y 429.826,Z 464.147,A -85,B 0,C 180,E1 -9648.683,E2 -9648.683} C_VEL
LIN {X 0,Y 431.019,Z 451.568,A -85,B 0,C 180,E1 -9649.899,E2 -9649.899} C_VEL
LIN {X 0,Y 432.145,Z 438.157,A -85,B 0,C 180,E1 -9650.964,E2 -9650.964} C_VEL
LIN {X 0,Y 433.27,Z 423.214,A -85,B 0,C 180,E1 -9651.905,E2 -9651.905} C_VEL
LIN {X 0,Y 434.152,Z 408.021,A -85,B 0,C 180,E1 -9652.637,E2 -9652.637} C_VEL
LIN {X 0,Y 434.79,Z 392.638,A -85,B 0,C 180,E1 -9653.172,E2 -9653.172} C_VEL
LIN {X 0,Y 435.234,Z 376.505,A -85,B 0,C 180,E1 -9653.524,E2 -9653.524} C_VEL
LIN {X 0,Y 436.803,Z 281.403,A -85,B 0,C 180,E1 -9655.117,E2 -9655.117} C_VEL
LIN {X 0,Y 437.315,Z 246.857,A -85,B 0,C 180,E1 -9655.701,E2 -9655.701} C_VEL
LIN {X 0,Y 434.777,Z 236.313,A -85,B 0,C 180,E1 -9656.053,E2 -9656.053} C_VEL
LIN {X 0,Y 428.205,Z 220.817,A -85,B 0,C 180,E1 -9656.786,E2 -9656.786} C_VEL
LIN {X 0,Y 425.318,Z 209.133,A -85,B 0,C 180,E1 -9659.308,E2 -9659.308} C_VEL
LIN {X 0,Y 425.28,Z 209.137,A -85,B 0,C 180,E1 -9662.562,E2 -9662.562} C_VEL
LIN {X 0,Y 425.298,Z 209.14,A -85,B 0,C 180,E1 -9665.335,E2 -9665.335} C_VEL
LIN {X 0,Y 425.309,Z 209.135,A -85,B 0,C 180,E1 -9668.896,E2 -9668.896} C_VEL
LIN {X 0,Y 425.288,Z 209.133,A -85,B 0,C 180,E1 -9671.958,E2 -9671.958} C_VEL
LIN {X 0,Y 425.282,Z 209.138,A -85,B 0,C 180,E1 -9675.282,E2 -9675.282} C_VEL
LIN {X 0,Y 425.299,Z 209.126,A -85,B 0,C 180,E1 -9678.624,E2 -9678.624} C_VEL
LIN {X 0,Y 425.317,Z 209.127,A -85,B 0,C 180,E1 -9681.103,E2 -9681.103} C_VEL
LIN {X 0,Y 425.295,Z 209.13,A -85,B 0,C 180,E1 -9684.664,E2 -9684.664} C_VEL
LIN {X 0,Y 425.26,Z 209.122,A -85,B 0,C 180,E1 -9688.073,E2 -9688.073} C_VEL
LIN {X 0,Y 425.331,Z 209.13,A -85,B 0,C 180,E1 -9691.368,E2 -9691.368} C_VEL
LIN {X 0,Y 425.288,Z 209.13,A -85,B 0,C 180,E1 -9694.554,E2 -9694.554} C_VEL
LIN {X 0,Y 425.28,Z 209.13,A -85,B 0,C 180,E1 -9697.661,E2 -9697.661} C_VEL
LIN {X 0,Y 425.354,Z 209.126,A -85,B 0,C 180,E1 -9700.704,E2 -9700.704} C_VEL
LIN {X 0,Y 425.38,Z 209.12,A -85,B 0,C 180,E1 -9703.688,E2 -9703.688} C_VEL
LIN {X 0,Y 425.404,Z 209.117,A -85,B 0,C 180,E1 -9707.598,E2 -9707.598} C_VEL
LIN {X 0,Y 425.434,Z 209.113,A -85,B 0,C 180,E1 -9711.45,E2 -9711.45} C_VEL
LIN {X 0,Y 425.545,Z 209.1,A -85,B 0,C 180,E1 -9714.313,E2 -9714.313} C_VEL
LIN {X 0,Y 425.567,Z 209.098,A -85,B 0,C 180,E1 -9718.107,E2 -9718.107} C_VEL
LIN {X 0,Y 425.695,Z 209.075,A -85,B 0,C 180,E1 -9720,E2 -9720} C_VEL
LIN {X 0,Y 425.549,Z 209.099,A -85,B 0,C 180,E1 -9722.84,E2 -9722.84} C_VEL
LIN {X 0,Y 425.521,Z 209.107,A -85,B 0,C 180,E1 -9726.639,E2 -9726.639} C_VEL
LIN {X 0,Y 425.393,Z 209.117,A -85,B 0,C 180,E1 -9729.509,E2 -9729.509} C_VEL
LIN {X 0,Y 425.385,Z 209.118,A -85,B 0,C 180,E1 -9732.904,E2 -9732.904} C_VEL
LIN {X 0,Y 425.361,Z 209.122,A -85,B 0,C 180,E1 -9736.609,E2 -9736.609} C_VEL
LIN {X 0,Y 425.32,Z 209.13,A -85,B 0,C 180,E1 -9739.636,E2 -9739.636} C_VEL
LIN {X 0,Y 425.299,Z 209.132,A -85,B 0,C 180,E1 -9743.365,E2 -9743.365} C_VEL
LIN {X 0,Y 425.34,Z 209.127,A -85,B 0,C 180,E1 -9746.845,E2 -9746.845} C_VEL
LIN {X 0,Y 425.311,Z 209.131,A -85,B 0,C 180,E1 -9749.718,E2 -9749.718} C_VEL
LIN {X 0,Y 425.277,Z 209.129,A -85,B 0,C 180,E1 -9753.048,E2 -9753.048} C_VEL
LIN {X 0,Y 425.276,Z 209.134,A -85,B 0,C 180,E1 -9755.929,E2 -9755.929} C_VEL
LIN {X 0,Y 425.288,Z 209.128,A -85,B 0,C 180,E1 -9759.043,E2 -9759.043} C_VEL
LIN {X 0,Y 425.269,Z 209.136,A -85,B 0,C 180,E1 -9762.654,E2 -9762.654} C_VEL
LIN {X 0,Y 425.256,Z 209.139,A -85,B 0,C 180,E1 -9766.045,E2 -9766.045} C_VEL
LIN {X 0,Y 425.3,Z 209.131,A -85,B 0,C 180,E1 -9768.626,E2 -9768.626} C_VEL
LIN {X 0,Y 425.318,Z 209.129,A -85,B 0,C 180,E1 -9771.105,E2 -9771.105} C_VEL
LIN {X 0,Y 425.297,Z 209.133,A -85,B 0,C 180,E1 -9774.665,E2 -9774.665} C_VEL
LIN {X 0,Y 425.288,Z 209.228,A -85,B 0,C 180,E1 -9777.382,E2 -9777.382} C_VEL
LIN {X 0,Y 429.056,Z 223.893,A -85,B 0,C 180,E1 -9780.244,E2 -9780.244} C_VEL
LIN {X 0,Y 431.331,Z 234.12,A -85,B 0,C 180,E1 -9782.144,E2 -9782.144} C_VEL
LIN {X 0,Y 430.75,Z 241.985,A -85,B 0,C 180,E1 -9783.432,E2 -9783.432} C_VEL
LIN {X 0,Y 436.93,Z 273.105,A -85,B 0,C 180,E1 -9784.39,E2 -9784.39} C_VEL
LIN {X 0,Y 435.258,Z 382.201,A -85,B 0,C 180,E1 -9786.224,E2 -9786.224} C_VEL
LIN {X 0,Y 434.702,Z 410.197,A -85,B 0,C 180,E1 -9786.729,E2 -9786.729} C_VEL
LIN {X 0,Y 433.991,Z 425.691,A -85,B 0,C 180,E1 -9787.194,E2 -9787.194} C_VEL
LIN {X 0,Y 433.118,Z 440.423,A -85,B 0,C 180,E1 -9787.826,E2 -9787.826} C_VEL
LIN {X 0,Y 432.025,Z 455.061,A -85,B 0,C 180,E1 -9788.655,E2 -9788.655} C_VEL
LIN {X 0,Y 430.915,Z 468.267,A -85,B 0,C 180,E1 -9789.598,E2 -9789.598} C_VEL
LIN {X 0,Y 429.646,Z 481.716,A -85,B 0,C 180,E1 -9790.78,E2 -9790.78} C_VEL
LIN {X 0,Y 428.503,Z 493.567,A -85,B 0,C 180,E1 -9792.04,E2 -9792.04} C_VEL
LIN {X 0,Y 427.369,Z 505.16,A -85,B 0,C 180,E1 -9793.521,E2 -9793.521} C_VEL
LIN {X 0,Y 426.347,Z 516.022,A -85,B 0,C 180,E1 -9795.197,E2 -9795.197} C_VEL
LIN {X 0,Y 425.467,Z 525.468,A -85,B 0,C 180,E1 -9796.958,E2 -9796.958} C_VEL
LIN {X 0,Y 425.066,Z 532.585,A -85,B 0,C 180,E1 -9798.556,E2 -9798.556} C_VEL
LIN {X 0,Y 424.514,Z 539.591,A -85,B 0,C 180,E1 -9800.471,E2 -9800.471} C_VEL
LIN {X 0,Y 424.306,Z 545.106,A -85,B 0,C 180,E1 -9802.386,E2 -9802.386} C_VEL
LIN {X 0,Y 424.139,Z 549.274,A -85,B 0,C 180,E1 -9804.294,E2 -9804.294} C_VEL
LIN {X 0,Y 424.051,Z 552.196,A -85,B 0,C 180,E1 -9806.199,E2 -9806.199} C_VEL
LIN {X 0,Y 424.124,Z 553.943,A -85,B 0,C 180,E1 -9808.101,E2 -9808.101} C_VEL
LIN {X 0,Y 424.081,Z 554.539,A -85,B 0,C 180,E1 -9810,E2 -9810} C_VEL
LIN {X 0,Y 424.124,Z 553.938,A -85,B 0,C 180,E1 -9811.899,E2 -9811.899} C_VEL
LIN {X 0,Y 424.051,Z 552.187,A -85,B 0,C 180,E1 -9813.801,E2 -9813.801} C_VEL
LIN {X 0,Y 424.15,Z 549.265,A -85,B 0,C 180,E1 -9815.706,E2 -9815.706} C_VEL
LIN {X 0,Y 424.306,Z 545.1,A -85,B 0,C 180,E1 -9817.614,E2 -9817.614} C_VEL
LIN {X 0,Y 424.514,Z 539.579,A -85,B 0,C 180,E1 -9819.529,E2 -9819.529} C_VEL
LIN {X 0,Y 425.067,Z 532.561,A -85,B 0,C 180,E1 -9821.444,E2 -9821.444} C_VEL
LIN {X 0,Y 425.602,Z 523.824,A -85,B 0,C 180,E1 -9823.366,E2 -9823.366} C_VEL
LIN {X 0,Y 426.474,Z 514.551,A -85,B 0,C 180,E1 -9825.043,E2 -9825.043} C_VEL
LIN {X 0,Y 427.384,Z 505.126,A -85,B 0,C 180,E1 -9826.479,E2 -9826.479} C_VEL
LIN {X 0,Y 428.524,Z 493.452,A -85,B 0,C 180,E1 -9827.968,E2 -9827.968} C_VEL
LIN {X 0,Y 429.746,Z 480.453,A -85,B 0,C 180,E1 -9829.339,E2 -9829.339} C_VEL
LIN {X 0,Y 430.885,Z 468.2,A -85,B 0,C 180,E1 -9830.404,E2 -9830.404} C_VEL
LIN {X 0,Y 432.014,Z 454.972,A -85,B 0,C 180,E1 -9831.345,E2 -9831.345} C_VEL
LIN {X 0,Y 433.129,Z 440.29,A -85,B 0,C 180,E1 -9832.175,E2 -9832.175} C_VEL
LIN {X 0,Y 433.988,Z 425.04,A -85,B 0,C 180,E1 -9832.828,E2 -9832.828} C_VEL
LIN {X 0,Y 434.682,Z 409.98,A -85,B 0,C 180,E1 -9833.272,E2 -9833.272} C_VEL
LIN {X 0,Y 435.376,Z 374.684,A -85,B 0,C 180,E1 -9833.895,E2 -9833.895} C_VEL
LIN {X 0,Y 436.986,Z 273.587,A -85,B 0,C 180,E1 -9835.591,E2 -9835.591} C_VEL
LIN {X 0,Y 430.739,Z 241.979,A -85,B 0,C 180,E1 -9836.561,E2 -9836.561} C_VEL
LIN {X 0,Y 431.353,Z 234.098,A -85,B 0,C 180,E1 -9837.851,E2 -9837.851} C_VEL
LIN {X 0,Y 428.672,Z 222.225,A -85,B 0,C 180,E1 -9840.062,E2 -9840.062} C_VEL
LIN {X 0,Y 425.287,Z 209.125,A -85,B 0,C 180,E1 -9842.654,E2 -9842.654} C_VEL
LIN {X 0,Y 425.281,Z 209.135,A -85,B 0,C 180,E1 -9845.929,E2 -9845.929} C_VEL
LIN {X 0,Y 425.307,Z 209.131,A -85,B 0,C 180,E1 -9849.045,E2 -9849.045} C_VEL
LIN {X 0,Y 425.311,Z 209.134,A -85,B 0,C 180,E1 -9851.961,E2 -9851.961} C_VEL
LIN {X 0,Y 425.28,Z 209.131,A -85,B 0,C 180,E1 -9855.282,E2 -9855.282} C_VEL
LIN {X 0,Y 425.298,Z 209.128,A -85,B 0,C 180,E1 -9858.624,E2 -9858.624} C_VEL
LIN {X 0,Y 425.316,Z 209.126,A -85,B 0,C 180,E1 -9861.103,E2 -9861.103} C_VEL
LIN {X 0,Y 425.294,Z 209.126,A -85,B 0,C 180,E1 -9864.664,E2 -9864.664} C_VEL
LIN {X 0,Y 425.266,Z 209.136,A -85,B 0,C 180,E1 -9868.073,E2 -9868.073} C_VEL
LIN {X 0,Y 425.33,Z 209.126,A -85,B 0,C 180,E1 -9871.368,E2 -9871.368} C_VEL
LIN {X 0,Y 425.287,Z 209.132,A -85,B 0,C 180,E1 -9874.554,E2 -9874.554} C_VEL
LIN {X 0,Y 425.28,Z 209.12,A -85,B 0,C 180,E1 -9877.661,E2 -9877.661} C_VEL
LIN {X 0,Y 425.354,Z 209.121,A -85,B 0,C 180,E1 -9880.704,E2 -9880.704} C_VEL
LIN {X 0,Y 425.38,Z 209.121,A -85,B 0,C 180,E1 -9883.688,E2 -9883.688} C_VEL
LIN {X 0,Y 425.404,Z 209.118,A -85,B 0,C 180,E1 -9887.598,E2 -9887.598} C_VEL
LIN {X 0,Y 425.434,Z 209.114,A -85,B 0,C 180,E1 -9891.45,E2 -9891.45} C_VEL
LIN {X 0,Y 425.546,Z 209.099,A -85,B 0,C 180,E1 -9894.313,E2 -9894.313} C_VEL
LIN {X 0,Y 425.567,Z 209.097,A -85,B 0,C 180,E1 -9898.107,E2 -9898.107} C_VEL
LIN {X 0,Y 425.695,Z 209.077,A -85,B 0,C 180,E1 -9900,E2 -9900} C_VEL
LIN {X 0,Y 425.549,Z 209.101,A -85,B 0,C 180,E1 -9902.84,E2 -9902.84} C_VEL
LIN {X 0,Y 425.523,Z 209.103,A -85,B 0,C 180,E1 -9906.65,E2 -9906.65} C_VEL
LIN {X 0,Y 425.394,Z 209.122,A -85,B 0,C 180,E1 -9909.51,E2 -9909.51} C_VEL
LIN {X 0,Y 425.386,Z 209.119,A -85,B 0,C 180,E1 -9912.905,E2 -9912.905} C_VEL
LIN {X 0,Y 425.353,Z 209.122,A -85,B 0,C 180,E1 -9916.605,E2 -9916.605} C_VEL
LIN {X 0,Y 425.321,Z 209.127,A -85,B 0,C 180,E1 -9919.636,E2 -9919.636} C_VEL
LIN {X 0,Y 425.28,Z 209.133,A -85,B 0,C 180,E1 -9922.339,E2 -9922.339} C_VEL
LIN {X 0,Y 425.288,Z 209.115,A -85,B 0,C 180,E1 -9925.446,E2 -9925.446} C_VEL
LIN {X 0,Y 425.331,Z 209.126,A -85,B 0,C 180,E1 -9928.632,E2 -9928.632} C_VEL
LIN {X 0,Y 425.26,Z 209.134,A -85,B 0,C 180,E1 -9931.927,E2 -9931.927} C_VEL
LIN {X 0,Y 425.295,Z 209.132,A -85,B 0,C 180,E1 -9935.336,E2 -9935.336} C_VEL
LIN {X 0,Y 425.304,Z 209.131,A -85,B 0,C 180,E1 -9938.898,E2 -9938.898} C_VEL
LIN {X 0,Y 425.286,Z 209.128,A -85,B 0,C 180,E1 -9941.959,E2 -9941.959} C_VEL
LIN {X 0,Y 425.287,Z 209.133,A -85,B 0,C 180,E1 -9945.283,E2 -9945.283} C_VEL
LIN {X 0,Y 425.273,Z 209.137,A -85,B 0,C 180,E1 -9948.622,E2 -9948.622} C_VEL
LIN {X 0,Y 425.309,Z 209.127,A -85,B 0,C 180,E1 -9951.104,E2 -9951.104} C_VEL
LIN {X 0,Y 425.297,Z 209.131,A -85,B 0,C 180,E1 -9954.665,E2 -9954.665} C_VEL
LIN {X 0,Y 425.264,Z 209.14,A -85,B 0,C 180,E1 -9958.074,E2 -9958.074} C_VEL
LIN {X 0,Y 425.304,Z 209.187,A -85,B 0,C 180,E1 -9960.814,E2 -9960.814} C_VEL
LIN {X 0,Y 428.213,Z 220.969,A -85,B 0,C 180,E1 -9963.329,E2 -9963.329} C_VEL
LIN {X 0,Y 435.377,Z 238.344,A -85,B 0,C 180,E1 -9964.119,E2 -9964.119} C_VEL
LIN {X 0,Y 437.305,Z 246.97,A -85,B 0,C 180,E1 -9964.397,E2 -9964.397} C_VEL
LIN {X 0,Y 435.635,Z 353.173,A -85,B 0,C 180,E1 -9966.183,E2 -9966.183} C_VEL
LIN {X 0,Y 434.994,Z 386.883,A -85,B 0,C 180,E1 -9966.777,E2 -9966.777} C_VEL
LIN {X 0,Y 434.44,Z 402.419,A -85,B 0,C 180,E1 -9967.243,E2 -9967.243} C_VEL
LIN {X 0,Y 433.692,Z 416.841,A -85,B 0,C 180,E1 -9967.859,E2 -9967.859} C_VEL
LIN {X 0,Y 432.648,Z 431.549,A -85,B 0,C 180,E1 -9968.687,E2 -9968.687} C_VEL
LIN {X 0,Y 431.61,Z 444.803,A -85,B 0,C 180,E1 -9969.632,E2 -9969.632} C_VEL
LIN {X 0,Y 430.379,Z 457.989,A -85,B 0,C 180,E1 -9970.786,E2 -9970.786} C_VEL
LIN {X 0,Y 429.288,Z 462.776,A -85,B 0,C 180,E1 -9971.23,E2 -9971.23} C_VEL
LIN {X 0,Y 425.788,Z 470.394,A -85,B 0,C 180,E1 -9971.948,E2 -9971.948} C_VEL
LIN {X 0,Y 422.307,Z 477.656,A -85,B 0,C 180,E1 -9972.732,E2 -9972.732} C_VEL
LIN {X 0,Y 421.245,Z 481.801,A -85,B 0,C 180,E1 -9973.273,E2 -9973.273} C_VEL
LIN {X 0,Y 420.109,Z 492.61,A -85,B 0,C 180,E1 -9974.972,E2 -9974.972} C_VEL
LIN {X 0,Y 419.056,Z 501.978,A -85,B 0,C 180,E1 -9976.756,E2 -9976.756} C_VEL
LIN {X 0,Y 418.527,Z 508.991,A -85,B 0,C 180,E1 -9978.375,E2 -9978.375} C_VEL
LIN {X 0,Y 417.883,Z 515.931,A -85,B 0,C 180,E1 -9980.318,E2 -9980.318} C_VEL
LIN {X 0,Y 417.509,Z 521.382,A -85,B 0,C 180,E1 -9982.261,E2 -9982.261} C_VEL
LIN {X 0,Y 417.285,Z 525.496,A -85,B 0,C 180,E1 -9984.2,E2 -9984.2} C_VEL
LIN {X 0,Y 417.066,Z 528.391,A -85,B 0,C 180,E1 -9986.135,E2 -9986.135} C_VEL
LIN {X 0,Y 417.077,Z 530.13,A -85,B 0,C 180,E1 -9988.069,E2 -9988.069} C_VEL
LIN {X 0,Y 417.002,Z 530.741,A -85,B 0,C 180,E1 -9990,E2 -9990} C_VEL
LIN {X 0,Y 417.078,Z 530.179,A -85,B 0,C 180,E1 -9991.931,E2 -9991.931} C_VEL
LIN {X 0,Y 417.065,Z 528.505,A -85,B 0,C 180,E1 -9993.865,E2 -9993.865} C_VEL
LIN {X 0,Y 417.268,Z 525.672,A -85,B 0,C 180,E1 -9995.8,E2 -9995.8} C_VEL
LIN {X 0,Y 417.479,Z 521.619,A -85,B 0,C 180,E1 -9997.74,E2 -9997.74} C_VEL
LIN {X 0,Y 417.871,Z 516.241,A -85,B 0,C 180,E1 -9999.682,E2 -9999.682} C_VEL
LIN {X 0,Y 418.514,Z 509.386,A -85,B 0,C 180,E1 -10001.625,E2 -10001.625} C_VEL
LIN {X 0,Y 419.174,Z 501.297,A -85,B 0,C 180,E1 -10003.481,E2 -10003.481} C_VEL
LIN {X 0,Y 420.204,Z 491.728,A -85,B 0,C 180,E1 -10005.273,E2 -10005.273} C_VEL
LIN {X 0,Y 421.188,Z 482.45,A -85,B 0,C 180,E1 -10006.728,E2 -10006.728} C_VEL
LIN {X 0,Y 422.367,Z 471.432,A -85,B 0,C 180,E1 -10008.179,E2 -10008.179} C_VEL
LIN {X 0,Y 423.589,Z 459.362,A -85,B 0,C 180,E1 -10009.505,E2 -10009.505} C_VEL
LIN {X 0,Y 424.869,Z 446.105,A -85,B 0,C 180,E1 -10010.706,E2 -10010.706} C_VEL
LIN {X 0,Y 425.948,Z 433.106,A -85,B 0,C 180,E1 -10011.665,E2 -10011.665} C_VEL
LIN {X 0,Y 426.994,Z 419.69,A -85,B 0,C 180,E1 -10012.454,E2 -10012.454} C_VEL
LIN {X 0,Y 427.761,Z 404.929,A -85,B 0,C 180,E1 -10013.132,E2 -10013.132} C_VEL
LIN {X 0,Y 428.379,Z 390.545,A -85,B 0,C 180,E1 -10013.603,E2 -10013.603} C_VEL
LIN {X 0,Y 428.815,Z 371.318,A -85,B 0,C 180,E1 -10013.995,E2 -10013.995} C_VEL
LIN {X 0,Y 430.397,Z 282.086,A -85,B 0,C 180,E1 -10015.508,E2 -10015.508} C_VEL
LIN {X 0,Y 430.876,Z 247.759,A -85,B 0,C 180,E1 -10016.101,E2 -10016.101} C_VEL
LIN {X 0,Y 428.697,Z 238.993,A -85,B 0,C 180,E1 -10016.405,E2 -10016.405} C_VEL
LIN {X 0,Y 421.014,Z 220.964,A -85,B 0,C 180,E1 -10017.294,E2 -10017.294} C_VEL
LIN {X 0,Y 418.266,Z 210.012,A -85,B 0,C 180,E1 -10019.713,E2 -10019.713} C_VEL
LIN {X 0,Y 418.247,Z 210.012,A -85,B 0,C 180,E1 -10023.676,E2 -10023.676} C_VEL
LIN {X 0,Y 418.243,Z 210.011,A -85,B 0,C 180,E1 -10027.223,E2 -10027.223} C_VEL
LIN {X 0,Y 418.247,Z 210.007,A -85,B 0,C 180,E1 -10029.681,E2 -10029.681} C_VEL
LIN {X 0,Y 418.229,Z 210.011,A -85,B 0,C 180,E1 -10032.321,E2 -10032.321} C_VEL
LIN {X 0,Y 418.234,Z 210.014,A -85,B 0,C 180,E1 -10035.108,E2 -10035.108} C_VEL
LIN {X 0,Y 418.252,Z 210.001,A -85,B 0,C 180,E1 -10037.768,E2 -10037.768} C_VEL
LIN {X 0,Y 418.262,Z 210.008,A -85,B 0,C 180,E1 -10040.616,E2 -10040.616} C_VEL
LIN {X 0,Y 418.241,Z 210.007,A -85,B 0,C 180,E1 -10043.975,E2 -10043.975} C_VEL
LIN {X 0,Y 418.252,Z 210.001,A -85,B 0,C 180,E1 -10047.155,E2 -10047.155} C_VEL
LIN {X 0,Y 418.268,Z 210.005,A -85,B 0,C 180,E1 -10050.838,E2 -10050.838} C_VEL
LIN {X 0,Y 418.263,Z 210.003,A -85,B 0,C 180,E1 -10054.095,E2 -10054.095} C_VEL
LIN {X 0,Y 418.231,Z 210.009,A -85,B 0,C 180,E1 -10057.263,E2 -10057.263} C_VEL
LIN {X 0,Y 418.275,Z 210.006,A -85,B 0,C 180,E1 -10060.364,E2 -10060.364} C_VEL
LIN {X 0,Y 418.309,Z 210.003,A -85,B 0,C 180,E1 -10063.404,E2 -10063.404} C_VEL
LIN {X 0,Y 418.338,Z 210.001,A -85,B 0,C 180,E1 -10066.999,E2 -10066.999} C_VEL
LIN {X 0,Y 418.333,Z 209.994,A -85,B 0,C 180,E1 -10070.328,E2 -10070.328} C_VEL
LIN {X 0,Y 418.484,Z 209.979,A -85,B 0,C 180,E1 -10073.249,E2 -10073.249} C_VEL
LIN {X 0,Y 418.332,Z 209.997,A -85,B 0,C 180,E1 -10075.181,E2 -10075.181} C_VEL
LIN {X 0,Y 418.536,Z 209.973,A -85,B 0,C 180,E1 -10078.075,E2 -10078.075} C_VEL
LIN {X 0,Y 418.665,Z 209.951,A -85,B 0,C 180,E1 -10080,E2 -10080} C_VEL
LIN {X 0,Y 418.502,Z 209.976,A -85,B 0,C 180,E1 -10082.888,E2 -10082.888} C_VEL
LIN {X 0,Y 418.484,Z 209.982,A -85,B 0,C 180,E1 -10086.751,E2 -10086.751} C_VEL
LIN {X 0,Y 418.333,Z 209.996,A -85,B 0,C 180,E1 -10089.671,E2 -10089.671} C_VEL
LIN {X 0,Y 418.338,Z 209.995,A -85,B 0,C 180,E1 -10093.001,E2 -10093.001} C_VEL
LIN {X 0,Y 418.312,Z 209.999,A -85,B 0,C 180,E1 -10096.739,E2 -10096.739} C_VEL
LIN {X 0,Y 418.262,Z 210.01,A -85,B 0,C 180,E1 -10099.791,E2 -10099.791} C_VEL
LIN {X 0,Y 418.23,Z 210.015,A -85,B 0,C 180,E1 -10102.736,E2 -10102.736} C_VEL
LIN {X 0,Y 418.263,Z 210.005,A -85,B 0,C 180,E1 -10105.904,E2 -10105.904} C_VEL
LIN {X 0,Y 418.267,Z 210.007,A -85,B 0,C 180,E1 -10109.162,E2 -10109.162} C_VEL
LIN {X 0,Y 418.253,Z 210.005,A -85,B 0,C 180,E1 -10112.845,E2 -10112.845} C_VEL
LIN {X 0,Y 418.239,Z 210.01,A -85,B 0,C 180,E1 -10116.239,E2 -10116.239} C_VEL
LIN {X 0,Y 418.244,Z 210.002,A -85,B 0,C 180,E1 -10119.683,E2 -10119.683} C_VEL
LIN {X 0,Y 418.224,Z 210.013,A -85,B 0,C 180,E1 -10122.322,E2 -10122.322} C_VEL
LIN {X 0,Y 418.23,Z 210.012,A -85,B 0,C 180,E1 -10125.109,E2 -10125.109} C_VEL
LIN {X 0,Y 418.252,Z 210.013,A -85,B 0,C 180,E1 -10127.769,E2 -10127.769} C_VEL
LIN {X 0,Y 418.263,Z 210.008,A -85,B 0,C 180,E1 -10130.618,E2 -10130.618} C_VEL
LIN {X 0,Y 418.243,Z 210.014,A -85,B 0,C 180,E1 -10133.977,E2 -10133.977} C_VEL
LIN {X 0,Y 418.252,Z 210.092,A -85,B 0,C 180,E1 -10136.959,E2 -10136.959} C_VEL
LIN {X 0,Y 422.128,Z 225.184,A -85,B 0,C 180,E1 -10139.968,E2 -10139.968} C_VEL
LIN {X 0,Y 424.464,Z 235.477,A -85,B 0,C 180,E1 -10141.922,E2 -10141.922} C_VEL
LIN {X 0,Y 424.08,Z 241.758,A -85,B 0,C 180,E1 -10142.977,E2 -10142.977} C_VEL
LIN {X 0,Y 430.53,Z 274.287,A -85,B 0,C 180,E1 -10144.006,E2 -10144.006} C_VEL
LIN {X 0,Y 428.796,Z 380.229,A -85,B 0,C 180,E1 -10145.811,E2 -10145.811} C_VEL
LIN {X 0,Y 428.203,Z 410.009,A -85,B 0,C 180,E1 -10146.354,E2 -10146.354} C_VEL
LIN {X 0,Y 427.485,Z 425.171,A -85,B 0,C 180,E1 -10146.813,E2 -10146.813} C_VEL
LIN {X 0,Y 426.561,Z 439.953,A -85,B 0,C 180,E1 -10147.451,E2 -10147.451} C_VEL
LIN {X 0,Y 425.563,Z 453.054,A -85,B 0,C 180,E1 -10148.188,E2 -10148.188} C_VEL
LIN {X 0,Y 424.347,Z 466.552,A -85,B 0,C 180,E1 -10149.141,E2 -10149.141} C_VEL
LIN {X 0,Y 423.059,Z 480.301,A -85,B 0,C 180,E1 -10150.343,E2 -10150.343} C_VEL
LIN {X 0,Y 421.751,Z 492.991,A -85,B 0,C 180,E1 -10151.697,E2 -10151.697} C_VEL
LIN {X 0,Y 420.524,Z 504.96,A -85,B 0,C 180,E1 -10153.245,E2 -10153.245} C_VEL
LIN {X 0,Y 419.394,Z 515.821,A -85,B 0,C 180,E1 -10154.946,E2 -10154.946} C_VEL
LIN {X 0,Y 418.632,Z 523.649,A -85,B 0,C 180,E1 -10156.407,E2 -10156.407} C_VEL
LIN {X 0,Y 418.038,Z 532.383,A -85,B 0,C 180,E1 -10158.361,E2 -10158.361} C_VEL
LIN {X 0,Y 417.437,Z 539.389,A -85,B 0,C 180,E1 -10160.308,E2 -10160.308} C_VEL
LIN {X 0,Y 417.228,Z 544.904,A -85,B 0,C 180,E1 -10162.256,E2 -10162.256} C_VEL
LIN {X 0,Y 417.058,Z 549.073,A -85,B 0,C 180,E1 -10164.197,E2 -10164.197} C_VEL
LIN {X 0,Y 416.966,Z 551.996,A -85,B 0,C 180,E1 -10166.134,E2 -10166.134} C_VEL
LIN {X 0,Y 417.051,Z 553.743,A -85,B 0,C 180,E1 -10168.069,E2 -10168.069} C_VEL
LIN {X 0,Y 417.001,Z 554.339,A -85,B 0,C 180,E1 -10170,E2 -10170} C_VEL
LIN {X 0,Y 417.051,Z 553.738,A -85,B 0,C 180,E1 -10171.931,E2 -10171.931} C_VEL
LIN {X 0,Y 416.966,Z 551.986,A -85,B 0,C 180,E1 -10173.866,E2 -10173.866} C_VEL
LIN {X 0,Y 417.068,Z 549.063,A -85,B 0,C 180,E1 -10175.803,E2 -10175.803} C_VEL
LIN {X 0,Y 417.229,Z 544.897,A -85,B 0,C 180,E1 -10177.744,E2 -10177.744} C_VEL
LIN {X 0,Y 417.437,Z 539.375,A -85,B 0,C 180,E1 -10179.692,E2 -10179.692} C_VEL
LIN {X 0,Y 418.037,Z 532.357,A -85,B 0,C 180,E1 -10181.639,E2 -10181.639} C_VEL
LIN {X 0,Y 418.631,Z 523.619,A -85,B 0,C 180,E1 -10183.593,E2 -10183.593} C_VEL
